   1:  PR[91,2] = PR[90,2] + 7.974;
   1:  PR[91,3] = PR[90,3] + 78.968;
   1:L PR[91] R[100]mm/sec CNT100;
   1:  PR[91,1] = PR[90,1] + 66.308;
   1:  PR[91,2] = PR[90,2] + 10.922;
   1:  PR[91,3] = PR[90,3] + 78.974;
   1:L PR[91] R[100]mm/sec CNT100;
   1:  PR[91,1] = PR[90,1] + 65.847;
   1:  PR[91,2] = PR[90,2] + 11.513;
   1:  PR[91,3] = PR[90,3] + 78.988;
   1:L PR[91] R[100]mm/sec CNT100;
   1:  PR[91,1] = PR[90,1] + 63.829;
   1:  PR[91,2] = PR[90,2] + 13.995;
   1:  PR[91,3] = PR[90,3] + 78.991;
   1:L PR[91] R[100]mm/sec CNT100;
   1:  PR[91,1] = PR[90,1] + 63.263;
   1:  PR[91,2] = PR[90,2] + 14.657;
   1:  PR[91,3] = PR[90,3] + 79.003;
   1:L PR[91] R[100]mm/sec CNT100;
   1:  PR[91,1] = PR[90,1] + 62.571;
   1:  PR[91,2] = PR[90,2] + 15.260;
   1:  PR[91,3] = PR[90,3] + 79.007;
   1:L PR[91] R[100]mm/sec CNT100;
   1:  PR[91,1] = PR[90,1] + 59.786;
   1:  PR[91,2] = PR[90,2] + 17.613;
   1:  PR[91,3] = PR[90,3] + 79.010;
   1:L PR[91] R[100]mm/sec CNT100;
   1:  PR[91,1] = PR[90,1] + 57.560;
   1:  PR[91,2] = PR[90,2] + 19.039;
   1:  PR[91,3] = PR[90,3] + 79.024;
   1:L PR[91] R[100]mm/sec CNT100;
   1:  PR[91,1] = PR[90,1] + 56.192;
   1:  PR[91,2] = PR[90,2] + 20.065;
   1:  PR[91,3] = PR[90,3] + 79.035;
   1:L PR[91] R[100]mm/sec CNT100;
   1:  PR[91,1] = PR[90,1] + 54.654;
   1:  PR[91,2] = PR[90,2] + 20.998;
   1:  PR[91,3] = PR[90,3] + 79.042;
   1:L PR[91] R[100]mm/sec CNT100;
   1:  PR[91,1] = PR[90,1] + 52.639;
   1:  PR[91,2] = PR[90,2] + 22.108;
   1:  PR[91,3] = PR[90,3] + 79.049;
   1:L PR[91] R[100]mm/sec CNT100;
   1:  PR[91,1] = PR[90,1] + 50.085;
   1:  PR[91,2] = PR[90,2] + 23.189;
   1:  PR[91,3] = PR[90,3] + 79.058;
   1:L PR[91] R[100]mm/sec CNT100;
   1:  PR[91,1] = PR[90,1] + 48.507;
   1:  PR[91,2] = PR[90,2] + 24.012;
   1:  PR[91,3] = PR[90,3] + 79.069;
   1:L PR[91] R[100]mm/sec CNT100;
   1:  PR[91,1] = PR[90,1] + 47.413;
   1:  PR[91,2] = PR[90,2] + 24.469;
   1:  PR[91,3] = PR[90,3] + 79.075;
   1:L PR[91] R[100]mm/sec CNT100;
   1:  PR[91,1] = PR[90,1] + 44.640;
   1:  PR[91,2] = PR[90,2] + 25.399;
   1:  PR[91,3] = PR[90,3] + 79.080;
   1:L PR[91] R[100]mm/sec CNT100;
   1:  PR[91,1] = PR[90,1] + 40.467;
   1:  PR[91,2] = PR[90,2] + 26.399;
   1:  PR[91,3] = PR[90,3] + 79.092;
   1:L PR[91] R[100]mm/sec CNT100;
   1:  PR[91,1] = PR[90,1] + 40.116;
   1:  PR[91,2] = PR[90,2] + 26.460;
   1:  PR[91,3] = PR[90,3] + 79.108;
   1:L PR[91] R[100]mm/sec CNT100;
   1:  PR[91,1] = PR[90,1] + 39.134;
   1:  PR[91,2] = PR[90,2] + 26.535;
   1:  PR[91,3] = PR[90,3] + 79.110;
   1:L PR[91] R[100]mm/sec CNT100;
   1:  PR[91,1] = PR[90,1] + 34.948;
   1:  PR[91,2] = PR[90,2] + 26.936;
   1:  PR[91,3] = PR[90,3] + 79.114;
   1:L PR[91] R[100]mm/sec CNT100;
   1:  PR[91,1] = PR[90,1] + 33.069;
   1:  PR[91,2] = PR[90,2] + 26.830;
   1:  PR[91,3] = PR[90,3] + 79.130;
   1:L PR[91] R[100]mm/sec CNT100;
   1:  PR[91,1] = PR[90,1] + 29.800;
   1:  PR[91,2] = PR[90,2] + 26.569;
   1:  PR[91,3] = PR[90,3] + 79.138;
   1:L PR[91] R[100]mm/sec CNT100;
   1:  PR[91,1] = PR[90,1] + 26.009;
   1:  PR[91,2] = PR[90,2] + 25.701;
   1:  PR[91,3] = PR[90,3] + 79.150;
   1:L PR[91] R[100]mm/sec CNT100;
   1:  PR[91,1] = PR[90,1] + 24.298;
   1:  PR[91,2] = PR[90,2] + 25.254;
   1:  PR[91,3] = PR[90,3] + 79.166;
   1:L PR[91] R[100]mm/sec CNT100;
   1:  PR[91,1] = PR[90,1] + 23.224;
   1:  PR[91,2] = PR[90,2] + 25.412;
   1:  PR[91,3] = PR[90,3] + 79.173;
   1:L PR[91] R[100]mm/sec CNT100;
   1:  PR[91,1] = PR[90,1] + 16.968;
   1:  PR[91,2] = PR[90,2] + 25.613;
   1:  PR[91,3] = PR[90,3] + 79.177;
   1:L PR[91] R[100]mm/sec CNT100;
   1:  PR[91,1] = PR[90,1] + 16.795;
   1:  PR[91,2] = PR[90,2] + 25.606;
   1:  PR[91,3] = PR[90,3] + 79.202;
   1:L PR[91] R[100]mm/sec CNT100;
   1:  PR[91,1] = PR[90,1] + 9.750;
   1:  PR[91,2] = PR[90,2] + 24.089;
   1:L PR[91] R[100]mm/sec CNT100;
   1:  PR[91,1] = PR[90,1] + 8.665;
   1:  PR[91,2] = PR[90,2] + 24.309;
   1:  PR[91,3] = PR[90,3] + 79.230;
   1:L PR[91] R[100]mm/sec CNT100;
   1:  PR[91,1] = PR[90,1] + 5.140;
   1:  PR[91,2] = PR[90,2] + 24.727;
   1:  PR[91,3] = PR[90,3] + 79.235;
   1:L PR[91] R[100]mm/sec CNT100;
   1:  PR[91,1] = PR[90,1] + 2.127;
   1:  PR[91,2] = PR[90,2] + 24.938;
   1:  PR[91,3] = PR[90,3] + 79.249;
   1:L PR[91] R[100]mm/sec CNT100;
   1:  PR[91,1] = PR[90,1] + -0.101;
   1:  PR[91,2] = PR[90,2] + 24.933;
   1:  PR[91,3] = PR[90,3] + 79.261;
   1:L PR[91] R[100]mm/sec CNT100;
   1:  PR[91,1] = PR[90,1] + -6.393;
   1:  PR[91,2] = PR[90,2] + 24.297;
   1:  PR[91,3] = PR[90,3] + 79.269;
   1:L PR[91] R[100]mm/sec CNT100;
   1:  PR[91,1] = PR[90,1] + -11.231;
   1:  PR[91,2] = PR[90,2] + 24.737;
   1:  PR[91,3] = PR[90,3] + 79.294;
   1:L PR[91] R[100]mm/sec CNT100;
   1:  PR[91,1] = PR[90,1] + -18.619;
   1:  PR[91,2] = PR[90,2] + 25.021;
   1:  PR[91,3] = PR[90,3] + 79.313;
   1:L PR[91] R[100]mm/sec CNT100;
   1:  PR[91,1] = PR[90,1] + -21.356;
   1:  PR[91,2] = PR[90,2] + 25.107;
   1:  PR[91,3] = PR[90,3] + 79.342;
   1:L PR[91] R[100]mm/sec CNT100;
   1:  PR[91,1] = PR[90,1] + -30.684;
   1:  PR[91,2] = PR[90,2] + 24.799;
   1:  PR[91,3] = PR[90,3] + 79.353;
   1:L PR[91] R[100]mm/sec CNT100;
   1:  PR[91,1] = PR[90,1] + -31.732;
   1:  PR[91,2] = PR[90,2] + 24.710;
   1:  PR[91,3] = PR[90,3] + 79.390;
   1:L PR[91] R[100]mm/sec CNT100;
   1:  PR[91,1] = PR[90,1] + -37.259;
   1:  PR[91,2] = PR[90,2] + 24.127;
   1:  PR[91,3] = PR[90,3] + 79.394;
   1:L PR[91] R[100]mm/sec CNT100;
   1:  PR[91,1] = PR[90,1] + -44.886;
   1:  PR[91,2] = PR[90,2] + 22.670;
   1:  PR[91,3] = PR[90,3] + 79.416;
   1:L PR[91] R[100]mm/sec CNT100;
   1:  PR[91,1] = PR[90,1] + -51.856;
   1:  PR[91,2] = PR[90,2] + 20.497;
   1:  PR[91,3] = PR[90,3] + 79.446;
   1:L PR[91] R[100]mm/sec CNT100;
   1:  PR[91,1] = PR[90,1] + -56.441;
   1:  PR[91,2] = PR[90,2] + 18.105;
   1:  PR[91,3] = PR[90,3] + 79.475;
   1:L PR[91] R[100]mm/sec CNT100;
   1:  PR[91] = PR[90];
   1:  PR[91,1] = PR[90,1] + -57.127;
   1:  PR[91,2] = PR[90,2] + 17.164;
   1:  PR[91,3] = PR[90,3] + 80.795;
   1:L PR[91] R[100]mm/sec CNT100;
   1:  PR[91,1] = PR[90,1] + -59.761;
   1:  PR[91,2] = PR[90,2] + 15.080;
   1:  PR[91,3] = PR[90,3] + 79.501;
   1:L PR[91] R[100]mm/sec CNT100;
   1:  PR[91,1] = PR[90,1] + -62.266;
   1:  PR[91,2] = PR[90,2] + 13.000;
   1:  PR[91,3] = PR[90,3] + 79.514;
   1:L PR[91] R[100]mm/sec CNT100;
   1:  PR[91,1] = PR[90,1] + -63.125;
   1:  PR[91,2] = PR[90,2] + 11.946;
   1:  PR[91,3] = PR[90,3] + 79.527;
   1:L PR[91] R[100]mm/sec CNT100;
   1:  PR[91,1] = PR[90,1] + -65.801;
   1:  PR[91,2] = PR[90,2] + 8.538;
   1:  PR[91,3] = PR[90,3] + 79.532;
   1:L PR[91] R[100]mm/sec CNT100;
   1:  PR[91,1] = PR[90,1] + -66.670;
   1:  PR[91,2] = PR[90,2] + 6.598;
   1:  PR[91,3] = PR[90,3] + 79.550;
   1:L PR[91] R[100]mm/sec CNT100;
   1:  PR[91,1] = PR[90,1] + -67.726;
   1:  PR[91,2] = PR[90,2] + 3.985;
   1:  PR[91,3] = PR[90,3] + 79.558;
   1:L PR[91] R[100]mm/sec CNT100;
   1:  PR[91,1] = PR[90,1] + -67.747;
   1:  PR[91,2] = PR[90,2] + 3.823;
   1:  PR[91,3] = PR[90,3] + 79.569;
   1:L PR[91] R[100]mm/sec CNT100;
   1:  PR[91,1] = PR[90,1] + -67.921;
   1:  PR[91,2] = PR[90,2] + 2.835;
   1:  PR[91,3] = PR[90,3] + 79.570;
   1:L PR[91] R[100]mm/sec CNT100;
   1:  PR[91,1] = PR[90,1] + -68.404;
   1:  PR[91,2] = PR[90,2] + -0.725;
   1:  PR[91,3] = PR[90,3] + 79.574;
   1:L PR[91] R[100]mm/sec CNT100;
   1:  PR[91,1] = PR[90,1] + -68.209;
   1:  PR[91,2] = PR[90,2] + -2.121;
   1:  PR[91,3] = PR[90,3] + 79.588;
   1:L PR[91] R[100]mm/sec CNT100;
   1:  PR[91,1] = PR[90,1] + -67.922;
   1:  PR[91,2] = PR[90,2] + -3.706;
   1:  PR[91,3] = PR[90,3] + 79.594;
   1:L PR[91] R[100]mm/sec CNT100;
   1:  PR[91,1] = PR[90,1] + -67.733;
   1:  PR[91,2] = PR[90,2] + -4.386;
   1:  PR[91,3] = PR[90,3] + 79.600;
   1:L PR[91] R[100]mm/sec CNT100;
   1:  PR[91,1] = PR[90,1] + -67.589;
   1:  PR[91,2] = PR[90,2] + -5.467;
   1:  PR[91,3] = PR[90,3] + 79.603;
   1:L PR[91] R[100]mm/sec CNT100;
   1:  PR[91,1] = PR[90,1] + -67.132;
   1:  PR[91,2] = PR[90,2] + -6.573;
   1:  PR[91,3] = PR[90,3] + 79.607;
   1:L PR[91] R[100]mm/sec CNT100;
   1:  PR[91,1] = PR[90,1] + -65.623;
   1:  PR[91,2] = PR[90,2] + -9.993;
   1:  PR[91,3] = PR[90,3] + 79.612;
   1:L PR[91] R[100]mm/sec CNT100;
   1:  PR[91,1] = PR[90,1] + -64.279;
   1:  PR[91,2] = PR[90,2] + -11.843;
   1:  PR[91,3] = PR[90,3] + 79.627;
   1:L PR[91] R[100]mm/sec CNT100;
   1:  PR[91,1] = PR[90,1] + -62.471;
   1:  PR[91,2] = PR[90,2] + -14.163;
   1:  PR[91,3] = PR[90,3] + 79.636;
   1:L PR[91] R[100]mm/sec CNT100;
   1:  PR[91,1] = PR[90,1] + -59.300;
   1:  PR[91,2] = PR[90,2] + -17.023;
   1:  PR[91,3] = PR[90,3] + 79.648;
   1:L PR[91] R[100]mm/sec CNT100;
   1:  PR[91,1] = PR[90,1] + -58.360;
   1:  PR[91,2] = PR[90,2] + -17.807;
   1:  PR[91,3] = PR[90,3] + 79.665;
   1:L PR[91] R[100]mm/sec CNT100;
   1:  PR[91,1] = PR[90,1] + -55.860;
   1:  PR[91,2] = PR[90,2] + -19.339;
   1:  PR[91,3] = PR[90,3] + 79.670;
   1:L PR[91] R[100]mm/sec CNT100;
   1:  PR[91,1] = PR[90,1] + -53.634;
   1:  PR[91,2] = PR[90,2] + -20.570;
   1:  PR[91,3] = PR[90,3] + 79.681;
   1:L PR[91] R[100]mm/sec CNT100;
   1:  PR[91,1] = PR[90,1] + -52.629;
   1:  PR[91,2] = PR[90,2] + -21.092;
   1:  PR[91,3] = PR[90,3] + 79.691;
   1:L PR[91] R[100]mm/sec CNT100;
   1:  PR[91,1] = PR[90,1] + -48.737;
   1:  PR[91,2] = PR[90,2] + -22.548;
   1:  PR[91,3] = PR[90,3] + 79.696;
   1:L PR[91] R[100]mm/sec CNT100;
   1:  PR[91,1] = PR[90,1] + -44.199;
   1:  PR[91,2] = PR[90,2] + -24.096;
   1:  PR[91,3] = PR[90,3] + 79.712;
   1:L PR[91] R[100]mm/sec CNT100;
   1:  PR[91,1] = PR[90,1] + -43.532;
   1:  PR[91,2] = PR[90,2] + -24.250;
   1:  PR[91,3] = PR[90,3] + 79.731;
   1:L PR[91] R[100]mm/sec CNT100;
   1:  PR[91,1] = PR[90,1] + -42.508;
   1:  PR[91,2] = PR[90,2] + -24.451;
   1:  PR[91,3] = PR[90,3] + 79.734;
   1:L PR[91] R[100]mm/sec CNT100;
   1:  PR[91,1] = PR[90,1] + -35.626;
   1:  PR[91,2] = PR[90,2] + -25.731;
   1:  PR[91,3] = PR[90,3] + 79.738;
   1:L PR[91] R[100]mm/sec CNT100;
   1:  PR[91,1] = PR[90,1] + -28.455;
   1:  PR[91,2] = PR[90,2] + -26.491;
   1:  PR[91,3] = PR[90,3] + 79.766;
   1:L PR[91] R[100]mm/sec CNT100;
   1:  PR[91,1] = PR[90,1] + -18.729;
   1:  PR[91,2] = PR[90,2] + -26.818;
   1:  PR[91,3] = PR[90,3] + 79.795;
   1:L PR[91] R[100]mm/sec CNT100;
   1:  PR[91,1] = PR[90,1] + -14.970;
   1:  PR[91,2] = PR[90,2] + -26.700;
   1:  PR[91,3] = PR[90,3] + 79.833;
   1:L PR[91] R[100]mm/sec CNT100;
   1:  PR[91,1] = PR[90,1] + -8.725;
   1:  PR[91,2] = PR[90,2] + -26.466;
   1:  PR[91,3] = PR[90,3] + 79.848;
   1:L PR[91] R[100]mm/sec CNT100;
   1:  PR[91,1] = PR[90,1] + -8.035;
   1:  PR[91,2] = PR[90,2] + -26.416;
   1:  PR[91,3] = PR[90,3] + 79.873;
   1:L PR[91] R[100]mm/sec CNT100;
   1:  PR[91,1] = PR[90,1] + -5.547;
   1:  PR[91,2] = PR[90,2] + -26.134;
   1:  PR[91,3] = PR[90,3] + 79.876;
   1:L PR[91] R[100]mm/sec CNT100;
   1:  PR[91,1] = PR[90,1] + -4.527;
   1:  PR[91,2] = PR[90,2] + -26.106;
   1:  PR[91,3] = PR[90,3] + 79.886;
   1:L PR[91] R[100]mm/sec CNT100;
   1:  PR[91,1] = PR[90,1] + -0.160;
   1:  PR[91,2] = PR[90,2] + -26.561;
   1:  PR[91,3] = PR[90,3] + 79.890;
   1:L PR[91] R[100]mm/sec CNT100;
   1:  PR[91,1] = PR[90,1] + 0.543;
   1:  PR[91,2] = PR[90,2] + -26.607;
   1:  PR[91,3] = PR[90,3] + 79.907;
   1:L PR[91] R[100]mm/sec CNT100;
   1:  PR[91,1] = PR[90,1] + 3.638;
   1:  PR[91,2] = PR[90,2] + -26.613;
   1:  PR[91,3] = PR[90,3] + 79.910;
   1:L PR[91] R[100]mm/sec CNT100;
   1:  PR[91,1] = PR[90,1] + 5.637;
   1:  PR[91,2] = PR[90,2] + -26.475;
   1:  PR[91,3] = PR[90,3] + 79.922;
   1:L PR[91] R[100]mm/sec CNT100;
   1:  PR[91,1] = PR[90,1] + 10.246;
   1:  PR[91,2] = PR[90,2] + -25.930;
   1:  PR[91,3] = PR[90,3] + 79.930;
   1:L PR[91] R[100]mm/sec CNT100;
   1:  PR[91,1] = PR[90,1] + 16.533;
   1:  PR[91,2] = PR[90,2] + -27.222;
   1:  PR[91,3] = PR[90,3] + 79.949;
   1:L PR[91] R[100]mm/sec CNT100;
   1:  PR[91,1] = PR[90,1] + 16.683;
   1:  PR[91,2] = PR[90,2] + -27.244;
   1:  PR[91,3] = PR[90,3] + 79.974;
   1:L PR[91] R[100]mm/sec CNT100;
   1:  PR[91,1] = PR[90,1] + 23.285;
   1:  PR[91,2] = PR[90,2] + -27.027;
   1:  PR[91,3] = PR[90,3] + 79.975;
   1:L PR[91] R[100]mm/sec CNT100;
   1:  PR[91,1] = PR[90,1] + 23.841;
   1:  PR[91,2] = PR[90,2] + -26.952;
   1:  PR[91,3] = PR[90,3] + 80.001;
   1:L PR[91] R[100]mm/sec CNT100;
   1:  PR[91,1] = PR[90,1] + 24.558;
   1:  PR[91,2] = PR[90,2] + -27.139;
   1:  PR[91,3] = PR[90,3] + 80.003;
   1:L PR[91] R[100]mm/sec CNT100;
   1:  PR[91,1] = PR[90,1] + 29.428;
   1:  PR[91,2] = PR[90,2] + -28.254;
   1:  PR[91,3] = PR[90,3] + 80.006;
   1:L PR[91] R[100]mm/sec CNT100;
   1:  PR[91,1] = PR[90,1] + 31.477;
   1:  PR[91,2] = PR[90,2] + -28.418;
   1:  PR[91,3] = PR[90,3] + 80.026;
   1:L PR[91] R[100]mm/sec CNT100;
   1:  PR[91,1] = PR[90,1] + 34.612;
   1:  PR[91,2] = PR[90,2] + -28.595;
   1:  PR[91,3] = PR[90,3] + 80.034;
   1:L PR[91] R[100]mm/sec CNT100;
   1:  PR[91,1] = PR[90,1] + 39.040;
   1:  PR[91,2] = PR[90,2] + -28.171;
   1:  PR[91,3] = PR[90,3] + 80.047;
   1:L PR[91] R[100]mm/sec CNT100;
   1:  PR[91,1] = PR[90,1] + 39.704;
   1:  PR[91,2] = PR[90,2] + -28.096;
   1:  PR[91,3] = PR[90,3] + 80.064;
   1:L PR[91] R[100]mm/sec CNT100;
   1:  PR[91,1] = PR[90,1] + 41.112;
   1:  PR[91,2] = PR[90,2] + -27.706;
   1:  PR[91,3] = PR[90,3] + 80.067;
   1:L PR[91] R[100]mm/sec CNT100;
   1:  PR[91,1] = PR[90,1] + 44.509;
   1:  PR[91,2] = PR[90,2] + -26.892;
   1:  PR[91,3] = PR[90,3] + 80.073;
   1:L PR[91] R[100]mm/sec CNT100;
   1:  PR[91,1] = PR[90,1] + 46.070;
   1:  PR[91,2] = PR[90,2] + -26.368;
   1:  PR[91,3] = PR[90,3] + 80.087;
   1:L PR[91] R[100]mm/sec CNT100;
   1:  PR[91,1] = PR[90,1] + 48.476;
   1:  PR[91,2] = PR[90,2] + -25.364;
   1:  PR[91,3] = PR[90,3] + 80.093;
   1:L PR[91] R[100]mm/sec CNT100;
   1:  PR[91,1] = PR[90,1] + 51.725;
   1:  PR[91,2] = PR[90,2] + -23.668;
   1:  PR[91,3] = PR[90,3] + 80.104;
   1:L PR[91] R[100]mm/sec CNT100;
   1:  PR[91,1] = PR[90,1] + 52.139;
   1:  PR[91,2] = PR[90,2] + -23.493;
   1:  PR[91,3] = PR[90,3] + 80.118;
   1:L PR[91] R[100]mm/sec CNT100;
   1:  PR[91,1] = PR[90,1] + 52.374;
   1:  PR[91,2] = PR[90,2] + -23.364;
   1:  PR[91,3] = PR[90,3] + 80.120;
   1:L PR[91] R[100]mm/sec CNT100;
   1:  PR[91,1] = PR[90,1] + 55.803;
   1:  PR[91,2] = PR[90,2] + -21.284;
   1:  PR[91,3] = PR[90,3] + 80.121;
   1:L PR[91] R[100]mm/sec CNT100;
   1:  PR[91,1] = PR[90,1] + 58.756;
   1:  PR[91,2] = PR[90,2] + -19.070;
   1:  PR[91,3] = PR[90,3] + 80.137;
   1:L PR[91] R[100]mm/sec CNT100;
   1:  PR[91,1] = PR[90,1] + 58.864;
   1:  PR[91,2] = PR[90,2] + -19.001;
   1:  PR[91,3] = PR[90,3] + 80.152;
   1:L PR[91] R[100]mm/sec CNT100;
   1:  PR[91,1] = PR[90,1] + 62.286;
   1:  PR[91,2] = PR[90,2] + -16.027;
   1:L PR[91] R[100]mm/sec CNT100;
   1:  PR[91,1] = PR[90,1] + 65.022;
   1:  PR[91,2] = PR[90,2] + -12.827;
   1:  PR[91,3] = PR[90,3] + 80.170;
   1:L PR[91] R[100]mm/sec CNT100;
   1:  PR[91,1] = PR[90,1] + 65.182;
   1:  PR[91,2] = PR[90,2] + -12.628;
   1:  PR[91,3] = PR[90,3] + 80.187;
   1:L PR[91] R[100]mm/sec CNT100;
   1:  PR[91,1] = PR[90,1] + 67.131;
   1:  PR[91,2] = PR[90,2] + -9.121;
   1:  PR[91,3] = PR[90,3] + 80.188;
   1:L PR[91] R[100]mm/sec CNT100;
   1:  PR[91,1] = PR[90,1] + 67.452;
   1:  PR[91,2] = PR[90,2] + -8.389;
   1:  PR[91,3] = PR[90,3] + 80.204;
   1:L PR[91] R[100]mm/sec CNT100;
   1:  PR[91,1] = PR[90,1] + 68.507;
   1:  PR[91,2] = PR[90,2] + -5.114;
   1:  PR[91,3] = PR[90,3] + 80.207;
   1:L PR[91] R[100]mm/sec CNT100;
   1:  PR[91,1] = PR[90,1] + 68.691;
   1:  PR[91,2] = PR[90,2] + -3.827;
   1:  PR[91,3] = PR[90,3] + 80.221;
   1:L PR[91] R[100]mm/sec CNT100;
   1:  PR[91,1] = PR[90,1] + 69.013;
   1:  PR[91,2] = PR[90,2] + -0.768;
   1:  PR[91,3] = PR[90,3] + 80.226;
   1:L PR[91] R[100]mm/sec CNT100;
   1:  PR[91,1] = PR[90,1] + 68.818;
   1:  PR[91,2] = PR[90,2] + 0.583;
   1:  PR[91,3] = PR[90,3] + 80.238;
   1:L PR[91] R[100]mm/sec CNT100;
   1:  PR[91,1] = PR[90,1] + 68.495;
   1:  PR[91,2] = PR[90,2] + 3.691;
   1:  PR[91,3] = PR[90,3] + 80.243;
   1:L PR[91] R[100]mm/sec CNT100;
   1:  PR[91,1] = PR[90,1] + 67.452;
   1:  PR[91,2] = PR[90,2] + 6.930;
   1:  PR[91,3] = PR[90,3] + 80.256;
   1:L PR[91] R[100]mm/sec CNT100;
   1:  PR[91,1] = PR[90,1] + 67.132;
   1:  PR[91,2] = PR[90,2] + 7.661;
   1:  PR[91,3] = PR[90,3] + 80.269;
   1:L PR[91] R[100]mm/sec CNT100;
   1:  PR[91,1] = PR[90,1] + 65.182;
   1:  PR[91,2] = PR[90,2] + 11.169;
   1:  PR[91,3] = PR[90,3] + 80.272;
   1:L PR[91] R[100]mm/sec CNT100;
   1:  PR[91,1] = PR[90,1] + 65.022;
   1:  PR[91,2] = PR[90,2] + 11.368;
   1:  PR[91,3] = PR[90,3] + 80.288;
   1:L PR[91] R[100]mm/sec CNT100;
   1:  PR[91,1] = PR[90,1] + 62.286;
   1:  PR[91,2] = PR[90,2] + 14.568;
   1:  PR[91,3] = PR[90,3] + 80.289;
   1:L PR[91] R[100]mm/sec CNT100;
   1:  PR[91,1] = PR[90,1] + 58.864;
   1:  PR[91,2] = PR[90,2] + 17.542;
   1:  PR[91,3] = PR[90,3] + 80.306;
   1:L PR[91] R[100]mm/sec CNT100;
   1:  PR[91,1] = PR[90,1] + 58.756;
   1:  PR[91,2] = PR[90,2] + 17.612;
   1:  PR[91,3] = PR[90,3] + 80.324;
   1:L PR[91] R[100]mm/sec CNT100;
   1:  PR[91,1] = PR[90,1] + 55.803;
   1:  PR[91,2] = PR[90,2] + 19.826;
   1:  PR[91,3] = PR[90,3] + 80.325;
   1:L PR[91] R[100]mm/sec CNT100;
   1:  PR[91,1] = PR[90,1] + 52.374;
   1:  PR[91,2] = PR[90,2] + 21.905;
   1:  PR[91,3] = PR[90,3] + 80.339;
   1:L PR[91] R[100]mm/sec CNT100;
   1:  PR[91,1] = PR[90,1] + 52.139;
   1:  PR[91,2] = PR[90,2] + 22.034;
   1:  PR[91,3] = PR[90,3] + 80.355;
   1:L PR[91] R[100]mm/sec CNT100;
   1:  PR[91,1] = PR[90,1] + 51.725;
   1:  PR[91,2] = PR[90,2] + 22.209;
   1:  PR[91,3] = PR[90,3] + 80.356;
   1:L PR[91] R[100]mm/sec CNT100;
   1:  PR[91,1] = PR[90,1] + 48.476;
   1:  PR[91,2] = PR[90,2] + 23.905;
   1:  PR[91,3] = PR[90,3] + 80.358;
   1:L PR[91] R[100]mm/sec CNT100;
   1:  PR[91,1] = PR[90,1] + 46.070;
   1:  PR[91,2] = PR[90,2] + 24.909;
   1:  PR[91,3] = PR[90,3] + 80.373;
   1:L PR[91] R[100]mm/sec CNT100;
   1:  PR[91,1] = PR[90,1] + 44.509;
   1:  PR[91,2] = PR[90,2] + 25.434;
   1:  PR[91,3] = PR[90,3] + 80.383;
   1:L PR[91] R[100]mm/sec CNT100;
   1:  PR[91,1] = PR[90,1] + 41.112;
   1:  PR[91,2] = PR[90,2] + 26.248;
   1:  PR[91,3] = PR[90,3] + 80.390;
   1:L PR[91] R[100]mm/sec CNT100;
   1:  PR[91,1] = PR[90,1] + 39.704;
   1:  PR[91,2] = PR[90,2] + 26.637;
   1:  PR[91,3] = PR[90,3] + 80.403;
   1:L PR[91] R[100]mm/sec CNT100;
   1:  PR[91,1] = PR[90,1] + 39.040;
   1:  PR[91,2] = PR[90,2] + 26.712;
   1:  PR[91,3] = PR[90,3] + 80.409;
   1:L PR[91] R[100]mm/sec CNT100;
   1:  PR[91,1] = PR[90,1] + 34.612;
   1:  PR[91,2] = PR[90,2] + 27.136;
   1:  PR[91,3] = PR[90,3] + 80.412;
   1:L PR[91] R[100]mm/sec CNT100;
   1:  PR[91,1] = PR[90,1] + 31.477;
   1:  PR[91,2] = PR[90,2] + 26.959;
   1:  PR[91,3] = PR[90,3] + 80.430;
   1:L PR[91] R[100]mm/sec CNT100;
   1:  PR[91,1] = PR[90,1] + 29.428;
   1:  PR[91,2] = PR[90,2] + 26.796;
   1:  PR[91,3] = PR[90,3] + 80.442;
   1:L PR[91] R[100]mm/sec CNT100;
   1:  PR[91,1] = PR[90,1] + 24.558;
   1:  PR[91,2] = PR[90,2] + 25.680;
   1:  PR[91,3] = PR[90,3] + 80.450;
   1:L PR[91] R[100]mm/sec CNT100;
   1:  PR[91,1] = PR[90,1] + 23.841;
   1:  PR[91,2] = PR[90,2] + 25.493;
   1:  PR[91,3] = PR[90,3] + 80.470;
   1:L PR[91] R[100]mm/sec CNT100;
   1:  PR[91,1] = PR[90,1] + 23.285;
   1:  PR[91,2] = PR[90,2] + 25.568;
   1:  PR[91,3] = PR[90,3] + 80.473;
   1:L PR[91] R[100]mm/sec CNT100;
   1:  PR[91,1] = PR[90,1] + 16.683;
   1:  PR[91,2] = PR[90,2] + 25.785;
   1:  PR[91,3] = PR[90,3] + 80.475;
   1:L PR[91] R[100]mm/sec CNT100;
   1:  PR[91,1] = PR[90,1] + 16.533;
   1:  PR[91,2] = PR[90,2] + 25.763;
   1:  PR[91,3] = PR[90,3] + 80.501;
   1:L PR[91] R[100]mm/sec CNT100;
   1:  PR[91,1] = PR[90,1] + 10.246;
   1:  PR[91,2] = PR[90,2] + 24.471;
   1:  PR[91,3] = PR[90,3] + 80.502;
   1:L PR[91] R[100]mm/sec CNT100;
   1:  PR[91,1] = PR[90,1] + 5.647;
   1:  PR[91,2] = PR[90,2] + 25.015;
   1:  PR[91,3] = PR[90,3] + 80.528;
   1:L PR[91] R[100]mm/sec CNT100;
   1:  PR[91,1] = PR[90,1] + 3.650;
   1:  PR[91,2] = PR[90,2] + 25.155;
   1:  PR[91,3] = PR[90,3] + 80.546;
   1:L PR[91] R[100]mm/sec CNT100;
   1:  PR[91,1] = PR[90,1] + 0.598;
   1:  PR[91,2] = PR[90,2] + 25.148;
   1:  PR[91,3] = PR[90,3] + 80.554;
   1:L PR[91] R[100]mm/sec CNT100;
   1:  PR[91,1] = PR[90,1] + -4.527;
   1:  PR[91,2] = PR[90,2] + 24.630;
   1:  PR[91,3] = PR[90,3] + 80.566;
   1:L PR[91] R[100]mm/sec CNT100;
   1:  PR[91,1] = PR[90,1] + -8.480;
   1:  PR[91,2] = PR[90,2] + 24.990;
   1:  PR[91,3] = PR[90,3] + 80.586;
   1:L PR[91] R[100]mm/sec CNT100;
   1:  PR[91,1] = PR[90,1] + -14.972;
   1:  PR[91,2] = PR[90,2] + 25.241;
   1:  PR[91,3] = PR[90,3] + 80.602;
   1:L PR[91] R[100]mm/sec CNT100;
   1:  PR[91,1] = PR[90,1] + -18.729;
   1:  PR[91,2] = PR[90,2] + 25.359;
   1:  PR[91,3] = PR[90,3] + 80.628;
   1:L PR[91] R[100]mm/sec CNT100;
   1:  PR[91,1] = PR[90,1] + -28.456;
   1:  PR[91,2] = PR[90,2] + 25.032;
   1:  PR[91,3] = PR[90,3] + 80.643;
   1:L PR[91] R[100]mm/sec CNT100;
   1:  PR[91,1] = PR[90,1] + -35.694;
   1:  PR[91,2] = PR[90,2] + 24.272;
   1:  PR[91,3] = PR[90,3] + 80.682;
   1:L PR[91] R[100]mm/sec CNT100;
   1:  PR[91,1] = PR[90,1] + -43.684;
   1:  PR[91,2] = PR[90,2] + 22.754;
   1:  PR[91,3] = PR[90,3] + 80.710;
   1:L PR[91] R[100]mm/sec CNT100;
   1:  PR[91,1] = PR[90,1] + -47.455;
   1:  PR[91,2] = PR[90,2] + 21.581;
   1:  PR[91,3] = PR[90,3] + 80.743;
   1:L PR[91] R[100]mm/sec CNT100;
   1:  PR[91,1] = PR[90,1] + -50.593;
   1:  PR[91,2] = PR[90,2] + 20.532;
   1:  PR[91,3] = PR[90,3] + 80.758;
   1:L PR[91] R[100]mm/sec CNT100;
   1:  PR[91,1] = PR[90,1] + -52.958;
   1:  PR[91,2] = PR[90,2] + 19.392;
   1:  PR[91,3] = PR[90,3] + 80.772;
   1:L PR[91] R[100]mm/sec CNT100;
   1:  PR[91,1] = PR[90,1] + -55.848;
   1:  PR[91,2] = PR[90,2] + 17.879;
   1:  PR[91,3] = PR[90,3] + 80.782;
   1:L PR[91] R[100]mm/sec CNT100;
   1:  PR[91] = PR[90];
   1:  PR[91,1] = PR[90,1] + -59.097;
   1:  PR[91,2] = PR[90,2] + 14.724;
   1:  PR[91,3] = PR[90,3] + 82.095;
   1:L PR[91] R[100]mm/sec CNT100;
   1:  PR[91,1] = PR[90,1] + -60.961;
   1:  PR[91,2] = PR[90,2] + 13.177;
   1:  PR[91,3] = PR[90,3] + 80.812;
   1:L PR[91] R[100]mm/sec CNT100;
   1:  PR[91,1] = PR[90,1] + -62.361;
   1:  PR[91,2] = PR[90,2] + 11.459;
   1:  PR[91,3] = PR[90,3] + 80.822;
   1:L PR[91] R[100]mm/sec CNT100;
   1:  PR[91,1] = PR[90,1] + -64.566;
   1:  PR[91,2] = PR[90,2] + 8.651;
   1:  PR[91,3] = PR[90,3] + 80.831;
   1:L PR[91] R[100]mm/sec CNT100;
   1:  PR[91,1] = PR[90,1] + -64.934;
   1:  PR[91,2] = PR[90,2] + 7.850;
   1:  PR[91,3] = PR[90,3] + 80.845;
   1:L PR[91] R[100]mm/sec CNT100;
   1:  PR[91,1] = PR[90,1] + -66.656;
   1:  PR[91,2] = PR[90,2] + 3.986;
   1:  PR[91,3] = PR[90,3] + 80.849;
   1:L PR[91] R[100]mm/sec CNT100;
   1:  PR[91,1] = PR[90,1] + -67.348;
   1:  PR[91,2] = PR[90,2] + -0.728;
   1:  PR[91,3] = PR[90,3] + 80.866;
   1:L PR[91] R[100]mm/sec CNT100;
   1:  PR[91,1] = PR[90,1] + -66.993;
   1:  PR[91,2] = PR[90,2] + -2.684;
   1:  PR[91,3] = PR[90,3] + 80.885;
   1:L PR[91] R[100]mm/sec CNT100;
   1:  PR[91,1] = PR[90,1] + -66.707;
   1:  PR[91,2] = PR[90,2] + -3.713;
   1:  PR[91,3] = PR[90,3] + 80.893;
   1:L PR[91] R[100]mm/sec CNT100;
   1:  PR[91,1] = PR[90,1] + -66.475;
   1:  PR[91,2] = PR[90,2] + -5.456;
   1:  PR[91,3] = PR[90,3] + 80.897;
   1:L PR[91] R[100]mm/sec CNT100;
   1:  PR[91,1] = PR[90,1] + -65.707;
   1:  PR[91,2] = PR[90,2] + -7.317;
   1:  PR[91,3] = PR[90,3] + 80.904;
   1:L PR[91] R[100]mm/sec CNT100;
   1:  PR[91,1] = PR[90,1] + -64.534;
   1:  PR[91,2] = PR[90,2] + -9.975;
   1:  PR[91,3] = PR[90,3] + 80.912;
   1:L PR[91] R[100]mm/sec CNT100;
   1:  PR[91,1] = PR[90,1] + -62.639;
   1:  PR[91,2] = PR[90,2] + -12.585;
   1:  PR[91,3] = PR[90,3] + 80.924;
   1:L PR[91] R[100]mm/sec CNT100;
   1:  PR[91,1] = PR[90,1] + -61.422;
   1:  PR[91,2] = PR[90,2] + -14.146;
   1:  PR[91,3] = PR[90,3] + 80.937;
   1:L PR[91] R[100]mm/sec CNT100;
   1:  PR[91,1] = PR[90,1] + -57.445;
   1:  PR[91,2] = PR[90,2] + -17.734;
   1:  PR[91,3] = PR[90,3] + 80.945;
   1:L PR[91] R[100]mm/sec CNT100;
   1:  PR[91,1] = PR[90,1] + -57.362;
   1:  PR[91,2] = PR[90,2] + -17.803;
   1:  PR[91,3] = PR[90,3] + 80.967;
   1:L PR[91] R[100]mm/sec CNT100;
   1:  PR[91,1] = PR[90,1] + -56.971;
   1:  PR[91,2] = PR[90,2] + -18.043;
   1:L PR[91] R[100]mm/sec CNT100;
   1:  PR[91,1] = PR[90,1] + -52.816;
   1:  PR[91,2] = PR[90,2] + -20.339;
   1:  PR[91,3] = PR[90,3] + 80.969;
   1:L PR[91] R[100]mm/sec CNT100;
   1:  PR[91,1] = PR[90,1] + -50.855;
   1:  PR[91,2] = PR[90,2] + -21.359;
   1:  PR[91,3] = PR[90,3] + 80.988;
   1:L PR[91] R[100]mm/sec CNT100;
   1:  PR[91,1] = PR[90,1] + -47.969;
   1:  PR[91,2] = PR[90,2] + -22.438;
   1:  PR[91,3] = PR[90,3] + 80.997;
   1:L PR[91] R[100]mm/sec CNT100;
   1:  PR[91,1] = PR[90,1] + -43.135;
   1:  PR[91,2] = PR[90,2] + -24.088;
   1:  PR[91,3] = PR[90,3] + 81.009;
   1:L PR[91] R[100]mm/sec CNT100;
   1:  PR[91,1] = PR[90,1] + -42.305;
   1:  PR[91,2] = PR[90,2] + -24.336;
   1:  PR[91,3] = PR[90,3] + 81.030;
   1:L PR[91] R[100]mm/sec CNT100;
   1:  PR[91,1] = PR[90,1] + -40.753;
   1:  PR[91,2] = PR[90,2] + -24.637;
   1:  PR[91,3] = PR[90,3] + 81.033;
   1:L PR[91] R[100]mm/sec CNT100;
   1:  PR[91,1] = PR[90,1] + -34.092;
   1:  PR[91,2] = PR[90,2] + -25.875;
   1:  PR[91,3] = PR[90,3] + 81.039;
   1:L PR[91] R[100]mm/sec CNT100;
   1:  PR[91,1] = PR[90,1] + -25.910;
   1:  PR[91,2] = PR[90,2] + -26.735;
   1:  PR[91,3] = PR[90,3] + 81.067;
   1:L PR[91] R[100]mm/sec CNT100;
   1:  PR[91,1] = PR[90,1] + -16.101;
   1:  PR[91,2] = PR[90,2] + -27.071;
   1:  PR[91,3] = PR[90,3] + 81.100;
   1:L PR[91] R[100]mm/sec CNT100;
   1:  PR[91,1] = PR[90,1] + -11.322;
   1:  PR[91,2] = PR[90,2] + -26.920;
   1:  PR[91,3] = PR[90,3] + 81.139;
   1:L PR[91] R[100]mm/sec CNT100;
   1:  PR[91,1] = PR[90,1] + -6.014;
   1:  PR[91,2] = PR[90,2] + -26.721;
   1:  PR[91,3] = PR[90,3] + 81.158;
   1:L PR[91] R[100]mm/sec CNT100;
   1:  PR[91,1] = PR[90,1] + -5.208;
   1:  PR[91,2] = PR[90,2] + -26.663;
   1:  PR[91,3] = PR[90,3] + 81.180;
   1:L PR[91] R[100]mm/sec CNT100;
   1:  PR[91,1] = PR[90,1] + -3.478;
   1:  PR[91,2] = PR[90,2] + -26.467;
   1:  PR[91,3] = PR[90,3] + 81.183;
   1:L PR[91] R[100]mm/sec CNT100;
   1:  PR[91,1] = PR[90,1] + -2.707;
   1:  PR[91,2] = PR[90,2] + -26.446;
   1:  PR[91,3] = PR[90,3] + 81.190;
   1:L PR[91] R[100]mm/sec CNT100;
   1:  PR[91,1] = PR[90,1] + 0.335;
   1:  PR[91,2] = PR[90,2] + -26.763;
   1:  PR[91,3] = PR[90,3] + 81.193;
   1:L PR[91] R[100]mm/sec CNT100;
   1:  PR[91,1] = PR[90,1] + 1.244;
   1:  PR[91,2] = PR[90,2] + -26.822;
   1:  PR[91,3] = PR[90,3] + 81.205;
   1:L PR[91] R[100]mm/sec CNT100;
   1:  PR[91,1] = PR[90,1] + 5.167;
   1:  PR[91,2] = PR[90,2] + -26.830;
   1:  PR[91,3] = PR[90,3] + 81.209;
   1:L PR[91] R[100]mm/sec CNT100;
   1:  PR[91,1] = PR[90,1] + 6.150;
   1:  PR[91,2] = PR[90,2] + -26.762;
   1:  PR[91,3] = PR[90,3] + 81.225;
   1:L PR[91] R[100]mm/sec CNT100;
   1:  PR[91,1] = PR[90,1] + 8.363;
   1:  PR[91,2] = PR[90,2] + -26.500;
   1:  PR[91,3] = PR[90,3] + 81.229;
   1:L PR[91] R[100]mm/sec CNT100;
   1:  PR[91,1] = PR[90,1] + 10.803;
   1:  PR[91,2] = PR[90,2] + -26.256;
   1:  PR[91,3] = PR[90,3] + 81.238;
   1:L PR[91] R[100]mm/sec CNT100;
   1:  PR[91,1] = PR[90,1] + 15.320;
   1:  PR[91,2] = PR[90,2] + -27.185;
   1:  PR[91,3] = PR[90,3] + 81.248;
   1:L PR[91] R[100]mm/sec CNT100;
   1:  PR[91,1] = PR[90,1] + 16.175;
   1:  PR[91,2] = PR[90,2] + -27.328;
   1:  PR[91,3] = PR[90,3] + 81.266;
   1:L PR[91] R[100]mm/sec CNT100;
   1:  PR[91,1] = PR[90,1] + 16.871;
   1:  PR[91,2] = PR[90,2] + -27.413;
   1:  PR[91,3] = PR[90,3] + 81.270;
   1:L PR[91] R[100]mm/sec CNT100;
   1:  PR[91,1] = PR[90,1] + 23.534;
   1:  PR[91,2] = PR[90,2] + -27.191;
   1:  PR[91,3] = PR[90,3] + 81.272;
   1:L PR[91] R[100]mm/sec CNT100;
   1:  PR[91,1] = PR[90,1] + 26.132;
   1:  PR[91,2] = PR[90,2] + -27.811;
   1:  PR[91,3] = PR[90,3] + 81.299;
   1:L PR[91] R[100]mm/sec CNT100;
   1:  PR[91,1] = PR[90,1] + 29.056;
   1:  PR[91,2] = PR[90,2] + -28.481;
   1:  PR[91,3] = PR[90,3] + 81.310;
   1:L PR[91] R[100]mm/sec CNT100;
   1:  PR[91,1] = PR[90,1] + 29.886;
   1:  PR[91,2] = PR[90,2] + -28.547;
   1:  PR[91,3] = PR[90,3] + 81.322;
   1:L PR[91] R[100]mm/sec CNT100;
   1:  PR[91,1] = PR[90,1] + 34.276;
   1:  PR[91,2] = PR[90,2] + -28.794;
   1:  PR[91,3] = PR[90,3] + 81.325;
   1:L PR[91] R[100]mm/sec CNT100;
   1:  PR[91,1] = PR[90,1] + 37.303;
   1:  PR[91,2] = PR[90,2] + -28.504;
   1:  PR[91,3] = PR[90,3] + 81.343;
   1:L PR[91] R[100]mm/sec CNT100;
   1:  PR[91,1] = PR[90,1] + 39.402;
   1:  PR[91,2] = PR[90,2] + -28.267;
   1:  PR[91,3] = PR[90,3] + 81.355;
   1:L PR[91] R[100]mm/sec CNT100;
   1:  PR[91,1] = PR[90,1] + 43.418;
   1:  PR[91,2] = PR[90,2] + -27.157;
   1:  PR[91,3] = PR[90,3] + 81.364;
   1:L PR[91] R[100]mm/sec CNT100;
   1:  PR[91,1] = PR[90,1] + 44.378;
   1:  PR[91,2] = PR[90,2] + -26.927;
   1:  PR[91,3] = PR[90,3] + 81.381;
   1:L PR[91] R[100]mm/sec CNT100;
   1:  PR[91,1] = PR[90,1] + 44.728;
   1:  PR[91,2] = PR[90,2] + -26.809;
   1:  PR[91,3] = PR[90,3] + 81.385;
   1:L PR[91] R[100]mm/sec CNT100;
   1:  PR[91,1] = PR[90,1] + 48.444;
   1:  PR[91,2] = PR[90,2] + -25.257;
   1:  PR[91,3] = PR[90,3] + 81.386;
   1:L PR[91] R[100]mm/sec CNT100;
   1:  PR[91,1] = PR[90,1] + 50.965;
   1:  PR[91,2] = PR[90,2] + -23.942;
   1:  PR[91,3] = PR[90,3] + 81.402;
   1:L PR[91] R[100]mm/sec CNT100;
   1:  PR[91,1] = PR[90,1] + 51.821;
   1:  PR[91,2] = PR[90,2] + -23.403;
   1:  PR[91,3] = PR[90,3] + 81.414;
   1:L PR[91] R[100]mm/sec CNT100;
   1:  PR[91,1] = PR[90,1] + 53.101;
   1:  PR[91,2] = PR[90,2] + -22.447;
   1:  PR[91,3] = PR[90,3] + 81.418;
   1:L PR[91] R[100]mm/sec CNT100;
   1:  PR[91,1] = PR[90,1] + 55.414;
   1:  PR[91,2] = PR[90,2] + -21.045;
   1:  PR[91,3] = PR[90,3] + 81.424;
   1:L PR[91] R[100]mm/sec CNT100;
   1:  PR[91,1] = PR[90,1] + 57.005;
   1:  PR[91,2] = PR[90,2] + -19.852;
   1:  PR[91,3] = PR[90,3] + 81.435;
   1:L PR[91] R[100]mm/sec CNT100;
   1:  PR[91,1] = PR[90,1] + 58.345;
   1:  PR[91,2] = PR[90,2] + -18.719;
   1:  PR[91,3] = PR[90,3] + 81.443;
   1:L PR[91] R[100]mm/sec CNT100;
   1:  PR[91,1] = PR[90,1] + 59.721;
   1:  PR[91,2] = PR[90,2] + -17.321;
   1:  PR[91,3] = PR[90,3] + 81.450;
   1:L PR[91] R[100]mm/sec CNT100;
   1:  PR[91,1] = PR[90,1] + 61.308;
   1:  PR[91,2] = PR[90,2] + -15.938;
   1:  PR[91,3] = PR[90,3] + 81.458;
   1:L PR[91] R[100]mm/sec CNT100;
   1:  PR[91,1] = PR[90,1] + 62.644;
   1:  PR[91,2] = PR[90,2] + -14.376;
   1:  PR[91,3] = PR[90,3] + 81.466;
   1:L PR[91] R[100]mm/sec CNT100;
   1:  PR[91,1] = PR[90,1] + 64.150;
   1:  PR[91,2] = PR[90,2] + -12.560;
   1:  PR[91,3] = PR[90,3] + 81.475;
   1:L PR[91] R[100]mm/sec CNT100;
   1:  PR[91,1] = PR[90,1] + 66.017;
   1:  PR[91,2] = PR[90,2] + -9.345;
   1:  PR[91,3] = PR[90,3] + 81.484;
   1:L PR[91] R[100]mm/sec CNT100;
   1:  PR[91,1] = PR[90,1] + 66.304;
   1:  PR[91,2] = PR[90,2] + -8.829;
   1:  PR[91,3] = PR[90,3] + 81.499;
   1:L PR[91] R[100]mm/sec CNT100;
   1:  PR[91,1] = PR[90,1] + 67.558;
   1:  PR[91,2] = PR[90,2] + -4.939;
   1:  PR[91,3] = PR[90,3] + 81.501;
   1:L PR[91] R[100]mm/sec CNT100;
   1:  PR[91,1] = PR[90,1] + 67.624;
   1:  PR[91,2] = PR[90,2] + -4.472;
   1:  PR[91,3] = PR[90,3] + 81.518;
   1:L PR[91] R[100]mm/sec CNT100;
   1:  PR[91,1] = PR[90,1] + 68.015;
   1:  PR[91,2] = PR[90,2] + -0.768;
   1:  PR[91,3] = PR[90,3] + 81.520;
   1:L PR[91] R[100]mm/sec CNT100;
   1:  PR[91,1] = PR[90,1] + 67.931;
   1:  PR[91,2] = PR[90,2] + -0.182;
   1:  PR[91,3] = PR[90,3] + 81.535;
   1:L PR[91] R[100]mm/sec CNT100;
   1:  PR[91,1] = PR[90,1] + 67.546;
   1:  PR[91,2] = PR[90,2] + 3.516;
   1:  PR[91,3] = PR[90,3] + 81.537;
   1:L PR[91] R[100]mm/sec CNT100;
   1:  PR[91,1] = PR[90,1] + 66.304;
   1:  PR[91,2] = PR[90,2] + 7.370;
   1:  PR[91,3] = PR[90,3] + 81.552;
   1:L PR[91] R[100]mm/sec CNT100;
   1:  PR[91,1] = PR[90,1] + 66.017;
   1:  PR[91,2] = PR[90,2] + 7.887;
   1:  PR[91,3] = PR[90,3] + 81.568;
   1:L PR[91] R[100]mm/sec CNT100;
   1:  PR[91,1] = PR[90,1] + 64.150;
   1:  PR[91,2] = PR[90,2] + 11.101;
   1:  PR[91,3] = PR[90,3] + 81.571;
   1:L PR[91] R[100]mm/sec CNT100;
   1:  PR[91,1] = PR[90,1] + 62.644;
   1:  PR[91,2] = PR[90,2] + 12.917;
   1:  PR[91,3] = PR[90,3] + 81.586;
   1:L PR[91] R[100]mm/sec CNT100;
   1:  PR[91,1] = PR[90,1] + 61.308;
   1:  PR[91,2] = PR[90,2] + 14.480;
   1:  PR[91,3] = PR[90,3] + 81.595;
   1:L PR[91] R[100]mm/sec CNT100;
   1:  PR[91,1] = PR[90,1] + 59.721;
   1:  PR[91,2] = PR[90,2] + 15.862;
   1:  PR[91,3] = PR[90,3] + 81.603;
   1:L PR[91] R[100]mm/sec CNT100;
   1:  PR[91,1] = PR[90,1] + 58.345;
   1:  PR[91,2] = PR[90,2] + 17.260;
   1:  PR[91,3] = PR[90,3] + 81.612;
   1:L PR[91] R[100]mm/sec CNT100;
   1:  PR[91,1] = PR[90,1] + 57.004;
   1:  PR[91,2] = PR[90,2] + 18.393;
   1:  PR[91,3] = PR[90,3] + 81.620;
   1:L PR[91] R[100]mm/sec CNT100;
   1:  PR[91,1] = PR[90,1] + 55.414;
   1:  PR[91,2] = PR[90,2] + 19.586;
   1:  PR[91,3] = PR[90,3] + 81.627;
   1:L PR[91] R[100]mm/sec CNT100;
   1:  PR[91,1] = PR[90,1] + 53.101;
   1:  PR[91,2] = PR[90,2] + 20.989;
   1:  PR[91,3] = PR[90,3] + 81.635;
   1:L PR[91] R[100]mm/sec CNT100;
   1:  PR[91,1] = PR[90,1] + 51.821;
   1:  PR[91,2] = PR[90,2] + 21.944;
   1:  PR[91,3] = PR[90,3] + 81.646;
   1:L PR[91] R[100]mm/sec CNT100;
   1:  PR[91,1] = PR[90,1] + 50.965;
   1:  PR[91,2] = PR[90,2] + 22.483;
   1:  PR[91,3] = PR[90,3] + 81.652;
   1:L PR[91] R[100]mm/sec CNT100;
   1:  PR[91,1] = PR[90,1] + 48.444;
   1:  PR[91,2] = PR[90,2] + 23.798;
   1:  PR[91,3] = PR[90,3] + 81.656;
   1:L PR[91] R[100]mm/sec CNT100;
   1:  PR[91,1] = PR[90,1] + 44.728;
   1:  PR[91,2] = PR[90,2] + 25.350;
   1:  PR[91,3] = PR[90,3] + 81.668;
   1:L PR[91] R[100]mm/sec CNT100;
   1:  PR[91,1] = PR[90,1] + 44.378;
   1:  PR[91,2] = PR[90,2] + 25.468;
   1:  PR[91,3] = PR[90,3] + 81.684;
   1:L PR[91] R[100]mm/sec CNT100;
   1:  PR[91,1] = PR[90,1] + 43.418;
   1:  PR[91,2] = PR[90,2] + 25.698;
   1:  PR[91,3] = PR[90,3] + 81.685;
   1:L PR[91] R[100]mm/sec CNT100;
   1:  PR[91,1] = PR[90,1] + 39.402;
   1:  PR[91,2] = PR[90,2] + 26.808;
   1:  PR[91,3] = PR[90,3] + 81.689;
   1:L PR[91] R[100]mm/sec CNT100;
   1:  PR[91,1] = PR[90,1] + 37.303;
   1:  PR[91,2] = PR[90,2] + 27.046;
   1:  PR[91,3] = PR[90,3] + 81.706;
   1:L PR[91] R[100]mm/sec CNT100;
   1:  PR[91,1] = PR[90,1] + 34.276;
   1:  PR[91,2] = PR[90,2] + 27.336;
   1:  PR[91,3] = PR[90,3] + 81.714;
   1:L PR[91] R[100]mm/sec CNT100;
   1:  PR[91,1] = PR[90,1] + 29.886;
   1:  PR[91,2] = PR[90,2] + 27.088;
   1:  PR[91,3] = PR[90,3] + 81.727;
   1:L PR[91] R[100]mm/sec CNT100;
   1:  PR[91,1] = PR[90,1] + 29.056;
   1:  PR[91,2] = PR[90,2] + 27.022;
   1:  PR[91,3] = PR[90,3] + 81.744;
   1:L PR[91] R[100]mm/sec CNT100;
   1:  PR[91,1] = PR[90,1] + 26.131;
   1:  PR[91,2] = PR[90,2] + 26.352;
   1:  PR[91,3] = PR[90,3] + 81.748;
   1:L PR[91] R[100]mm/sec CNT100;
   1:  PR[91,1] = PR[90,1] + 23.532;
   1:  PR[91,2] = PR[90,2] + 25.732;
   1:  PR[91,3] = PR[90,3] + 81.760;
   1:L PR[91] R[100]mm/sec CNT100;
   1:  PR[91,1] = PR[90,1] + 17.636;
   1:  PR[91,2] = PR[90,2] + 25.942;
   1:  PR[91,3] = PR[90,3] + 81.770;
   1:L PR[91] R[100]mm/sec CNT100;
   1:  PR[91,1] = PR[90,1] + 16.885;
   1:  PR[91,2] = PR[90,2] + 25.956;
   1:  PR[91,3] = PR[90,3] + 81.794;
   1:L PR[91] R[100]mm/sec CNT100;
   1:  PR[91,1] = PR[90,1] + 16.176;
   1:  PR[91,2] = PR[90,2] + 25.869;
   1:  PR[91,3] = PR[90,3] + 81.797;
   1:L PR[91] R[100]mm/sec CNT100;
   1:  PR[91,1] = PR[90,1] + 15.321;
   1:  PR[91,2] = PR[90,2] + 25.726;
   1:  PR[91,3] = PR[90,3] + 81.800;
   1:L PR[91] R[100]mm/sec CNT100;
   1:  PR[91,1] = PR[90,1] + 10.804;
   1:  PR[91,2] = PR[90,2] + 24.798;
   1:  PR[91,3] = PR[90,3] + 81.804;
   1:L PR[91] R[100]mm/sec CNT100;
   1:  PR[91,1] = PR[90,1] + 8.361;
   1:  PR[91,2] = PR[90,2] + 25.041;
   1:  PR[91,3] = PR[90,3] + 81.822;
   1:L PR[91] R[100]mm/sec CNT100;
   1:  PR[91,1] = PR[90,1] + 6.155;
   1:  PR[91,2] = PR[90,2] + 25.303;
   1:  PR[91,3] = PR[90,3] + 81.832;
   1:L PR[91] R[100]mm/sec CNT100;
   1:  PR[91,1] = PR[90,1] + 5.173;
   1:  PR[91,2] = PR[90,2] + 25.372;
   1:  PR[91,3] = PR[90,3] + 81.841;
   1:L PR[91] R[100]mm/sec CNT100;
   1:  PR[91,1] = PR[90,1] + 1.298;
   1:  PR[91,2] = PR[90,2] + 25.364;
   1:  PR[91,3] = PR[90,3] + 81.845;
   1:L PR[91] R[100]mm/sec CNT100;
   1:  PR[91,1] = PR[90,1] + -2.664;
   1:  PR[91,2] = PR[90,2] + 24.963;
   1:  PR[91,3] = PR[90,3] + 81.860;
   1:L PR[91] R[100]mm/sec CNT100;
   1:  PR[91,1] = PR[90,1] + -5.173;
   1:  PR[91,2] = PR[90,2] + 25.202;
   1:  PR[91,3] = PR[90,3] + 81.876;
   1:L PR[91] R[100]mm/sec CNT100;
   1:  PR[91,1] = PR[90,1] + -5.712;
   1:  PR[91,2] = PR[90,2] + 25.242;
   1:  PR[91,3] = PR[90,3] + 81.887;
   1:L PR[91] R[100]mm/sec CNT100;
   1:  PR[91,1] = PR[90,1] + -11.323;
   1:  PR[91,2] = PR[90,2] + 25.461;
   1:  PR[91,3] = PR[90,3] + 81.889;
   1:L PR[91] R[100]mm/sec CNT100;
   1:  PR[91,1] = PR[90,1] + -16.101;
   1:  PR[91,2] = PR[90,2] + 25.612;
   1:  PR[91,3] = PR[90,3] + 81.911;
   1:L PR[91] R[100]mm/sec CNT100;
   1:  PR[91,1] = PR[90,1] + -25.910;
   1:  PR[91,2] = PR[90,2] + 25.277;
   1:  PR[91,3] = PR[90,3] + 81.930;
   1:L PR[91] R[100]mm/sec CNT100;
   1:  PR[91,1] = PR[90,1] + -34.129;
   1:  PR[91,2] = PR[90,2] + 24.417;
   1:  PR[91,3] = PR[90,3] + 81.970;
   1:L PR[91] R[100]mm/sec CNT100;
   1:  PR[91,1] = PR[90,1] + -42.483;
   1:  PR[91,2] = PR[90,2] + 22.838;
   1:  PR[91,3] = PR[90,3] + 82.003;
   1:L PR[91] R[100]mm/sec CNT100;
   1:  PR[91,1] = PR[90,1] + -43.134;
   1:  PR[91,2] = PR[90,2] + 22.635;
   1:  PR[91,3] = PR[90,3] + 82.037;
   1:L PR[91] R[100]mm/sec CNT100;
   1:  PR[91,1] = PR[90,1] + -49.319;
   1:  PR[91,2] = PR[90,2] + 20.568;
   1:  PR[91,3] = PR[90,3] + 82.040;
   1:L PR[91] R[100]mm/sec CNT100;
   1:  PR[91,1] = PR[90,1] + -54.015;
   1:  PR[91,2] = PR[90,2] + 18.303;
   1:  PR[91,3] = PR[90,3] + 82.066;
   1:L PR[91] R[100]mm/sec CNT100;
   1:  PR[91,1] = PR[90,1] + -55.257;
   1:  PR[91,2] = PR[90,2] + 17.653;
   1:  PR[91,3] = PR[90,3] + 82.087;
   1:L PR[91] R[100]mm/sec CNT100;
   1:  PR[91,1] = PR[90,1] + -55.728;
   1:  PR[91,2] = PR[90,2] + 17.390;
   1:  PR[91,3] = PR[90,3] + 82.093;
   1:L PR[91] R[100]mm/sec CNT100;
   1:  PR[91] = PR[90];
   1:  PR[91,1] = PR[90,1] + -58.434;
   1:  PR[91,2] = PR[90,2] + 14.368;
   1:  PR[91,3] = PR[90,3] + 83.395;
   1:L PR[91] R[100]mm/sec CNT100;
   1:  PR[91,1] = PR[90,1] + -59.656;
   1:  PR[91,2] = PR[90,2] + 13.353;
   1:  PR[91,3] = PR[90,3] + 82.114;
   1:L PR[91] R[100]mm/sec CNT100;
   1:  PR[91,1] = PR[90,1] + -61.596;
   1:  PR[91,2] = PR[90,2] + 10.973;
   1:  PR[91,3] = PR[90,3] + 82.120;
   1:L PR[91] R[100]mm/sec CNT100;
   1:  PR[91,1] = PR[90,1] + -63.324;
   1:  PR[91,2] = PR[90,2] + 8.772;
   1:  PR[91,3] = PR[90,3] + 82.133;
   1:L PR[91] R[100]mm/sec CNT100;
   1:  PR[91,1] = PR[90,1] + -64.034;
   1:  PR[91,2] = PR[90,2] + 7.229;
   1:  PR[91,3] = PR[90,3] + 82.144;
   1:L PR[91] R[100]mm/sec CNT100;
   1:  PR[91,1] = PR[90,1] + -65.452;
   1:  PR[91,2] = PR[90,2] + 4.047;
   1:  PR[91,3] = PR[90,3] + 82.151;
   1:L PR[91] R[100]mm/sec CNT100;
   1:  PR[91,1] = PR[90,1] + -66.056;
   1:  PR[91,2] = PR[90,2] + -0.072;
   1:  PR[91,3] = PR[90,3] + 82.165;
   1:L PR[91] R[100]mm/sec CNT100;
   1:  PR[91,1] = PR[90,1] + -66.225;
   1:  PR[91,2] = PR[90,2] + -0.783;
   1:  PR[91,3] = PR[90,3] + 82.182;
   1:L PR[91] R[100]mm/sec CNT100;
   1:  PR[91,1] = PR[90,1] + -66.065;
   1:  PR[91,2] = PR[90,2] + -1.662;
   1:  PR[91,3] = PR[90,3] + 82.185;
   1:L PR[91] R[100]mm/sec CNT100;
   1:  PR[91,1] = PR[90,1] + -65.682;
   1:  PR[91,2] = PR[90,2] + -3.041;
   1:  PR[91,3] = PR[90,3] + 82.189;
   1:L PR[91] R[100]mm/sec CNT100;
   1:  PR[91,1] = PR[90,1] + -65.361;
   1:  PR[91,2] = PR[90,2] + -5.445;
   1:  PR[91,3] = PR[90,3] + 82.195;
   1:L PR[91] R[100]mm/sec CNT100;
   1:  PR[91,1] = PR[90,1] + -64.283;
   1:  PR[91,2] = PR[90,2] + -8.061;
   1:  PR[91,3] = PR[90,3] + 82.205;
   1:L PR[91] R[100]mm/sec CNT100;
   1:  PR[91,1] = PR[90,1] + -63.445;
   1:  PR[91,2] = PR[90,2] + -9.958;
   1:  PR[91,3] = PR[90,3] + 82.216;
   1:L PR[91] R[100]mm/sec CNT100;
   1:  PR[91,1] = PR[90,1] + -60.998;
   1:  PR[91,2] = PR[90,2] + -13.327;
   1:  PR[91,3] = PR[90,3] + 82.225;
   1:L PR[91] R[100]mm/sec CNT100;
   1:  PR[91,1] = PR[90,1] + -60.372;
   1:  PR[91,2] = PR[90,2] + -14.130;
   1:  PR[91,3] = PR[90,3] + 82.242;
   1:L PR[91] R[100]mm/sec CNT100;
   1:  PR[91,1] = PR[90,1] + -57.789;
   1:  PR[91,2] = PR[90,2] + -16.460;
   1:  PR[91,3] = PR[90,3] + 82.246;
   1:L PR[91] R[100]mm/sec CNT100;
   1:  PR[91,1] = PR[90,1] + -56.374;
   1:  PR[91,2] = PR[90,2] + -17.599;
   1:  PR[91,3] = PR[90,3] + 82.260;
   1:L PR[91] R[100]mm/sec CNT100;
   1:  PR[91,1] = PR[90,1] + -55.956;
   1:  PR[91,2] = PR[90,2] + -17.921;
   1:  PR[91,3] = PR[90,3] + 82.267;
   1:L PR[91] R[100]mm/sec CNT100;
   1:  PR[91,1] = PR[90,1] + -51.998;
   1:  PR[91,2] = PR[90,2] + -20.108;
   1:  PR[91,3] = PR[90,3] + 82.269;
   1:L PR[91] R[100]mm/sec CNT100;
   1:  PR[91,1] = PR[90,1] + -49.080;
   1:  PR[91,2] = PR[90,2] + -21.626;
   1:  PR[91,3] = PR[90,3] + 82.288;
   1:L PR[91] R[100]mm/sec CNT100;
   1:  PR[91,1] = PR[90,1] + -47.201;
   1:  PR[91,2] = PR[90,2] + -22.328;
   1:  PR[91,3] = PR[90,3] + 82.301;
   1:L PR[91] R[100]mm/sec CNT100;
   1:  PR[91,1] = PR[90,1] + -43.991;
   1:  PR[91,2] = PR[90,2] + -23.424;
   1:  PR[91,3] = PR[90,3] + 82.309;
   1:L PR[91] R[100]mm/sec CNT100;
   1:  PR[91,1] = PR[90,1] + -41.563;
   1:  PR[91,2] = PR[90,2] + -24.162;
   1:  PR[91,3] = PR[90,3] + 82.323;
   1:L PR[91] R[100]mm/sec CNT100;
   1:  PR[91,1] = PR[90,1] + -40.306;
   1:  PR[91,2] = PR[90,2] + -24.526;
   1:  PR[91,3] = PR[90,3] + 82.334;
   1:L PR[91] R[100]mm/sec CNT100;
   1:  PR[91,1] = PR[90,1] + -32.552;
   1:  PR[91,2] = PR[90,2] + -26.021;
   1:  PR[91,3] = PR[90,3] + 82.339;
   1:L PR[91] R[100]mm/sec CNT100;
   1:  PR[91,1] = PR[90,1] + -23.360;
   1:  PR[91,2] = PR[90,2] + -26.980;
   1:  PR[91,3] = PR[90,3] + 82.371;
   1:L PR[91] R[100]mm/sec CNT100;
   1:  PR[91,1] = PR[90,1] + -20.690;
   1:  PR[91,2] = PR[90,2] + -27.083;
   1:  PR[91,3] = PR[90,3] + 82.409;
   1:L PR[91] R[100]mm/sec CNT100;
   1:  PR[91,1] = PR[90,1] + -13.475;
   1:  PR[91,2] = PR[90,2] + -27.323;
   1:  PR[91,3] = PR[90,3] + 82.419;
   1:L PR[91] R[100]mm/sec CNT100;
   1:  PR[91,1] = PR[90,1] + -7.674;
   1:  PR[91,2] = PR[90,2] + -27.140;
   1:  PR[91,3] = PR[90,3] + 82.449;
   1:L PR[91] R[100]mm/sec CNT100;
   1:  PR[91,1] = PR[90,1] + -3.302;
   1:  PR[91,2] = PR[90,2] + -26.977;
   1:  PR[91,3] = PR[90,3] + 82.472;
   1:L PR[91] R[100]mm/sec CNT100;
   1:  PR[91,1] = PR[90,1] + -2.382;
   1:  PR[91,2] = PR[90,2] + -26.911;
   1:  PR[91,3] = PR[90,3] + 82.490;
   1:L PR[91] R[100]mm/sec CNT100;
   1:  PR[91,1] = PR[90,1] + -1.409;
   1:  PR[91,2] = PR[90,2] + -26.800;
   1:  PR[91,3] = PR[90,3] + 82.494;
   1:L PR[91] R[100]mm/sec CNT100;
   1:  PR[91,1] = PR[90,1] + -0.887;
   1:  PR[91,2] = PR[90,2] + -26.786;
   1:  PR[91,3] = PR[90,3] + 82.498;
   1:L PR[91] R[100]mm/sec CNT100;
   1:  PR[91,1] = PR[90,1] + 0.830;
   1:  PR[91,2] = PR[90,2] + -26.965;
   1:  PR[91,3] = PR[90,3] + 82.500;
   1:L PR[91] R[100]mm/sec CNT100;
   1:  PR[91,1] = PR[90,1] + 1.945;
   1:  PR[91,2] = PR[90,2] + -27.037;
   1:  PR[91,3] = PR[90,3] + 82.507;
   1:L PR[91] R[100]mm/sec CNT100;
   1:  PR[91,1] = PR[90,1] + 6.664;
   1:  PR[91,2] = PR[90,2] + -27.047;
   1:  PR[91,3] = PR[90,3] + 82.512;
   1:L PR[91] R[100]mm/sec CNT100;
   1:  PR[91,1] = PR[90,1] + 11.342;
   1:  PR[91,2] = PR[90,2] + -26.579;
   1:  PR[91,3] = PR[90,3] + 82.531;
   1:L PR[91] R[100]mm/sec CNT100;
   1:  PR[91,1] = PR[90,1] + 14.086;
   1:  PR[91,2] = PR[90,2] + -27.144;
   1:  PR[91,3] = PR[90,3] + 82.550;
   1:L PR[91] R[100]mm/sec CNT100;
   1:  PR[91,1] = PR[90,1] + 15.681;
   1:  PR[91,2] = PR[90,2] + -27.410;
   1:  PR[91,3] = PR[90,3] + 82.561;
   1:L PR[91] R[100]mm/sec CNT100;
   1:  PR[91,1] = PR[90,1] + 17.081;
   1:  PR[91,2] = PR[90,2] + -27.582;
   1:  PR[91,3] = PR[90,3] + 82.568;
   1:L PR[91] R[100]mm/sec CNT100;
   1:  PR[91,1] = PR[90,1] + 21.770;
   1:  PR[91,2] = PR[90,2] + -27.421;
   1:  PR[91,3] = PR[90,3] + 82.574;
   1:L PR[91] R[100]mm/sec CNT100;
   1:  PR[91,1] = PR[90,1] + 23.238;
   1:  PR[91,2] = PR[90,2] + -27.394;
   1:  PR[91,3] = PR[90,3] + 82.593;
   1:L PR[91] R[100]mm/sec CNT100;
   1:  PR[91,1] = PR[90,1] + 28.693;
   1:  PR[91,2] = PR[90,2] + -28.697;
   1:  PR[91,3] = PR[90,3] + 82.599;
   1:L PR[91] R[100]mm/sec CNT100;
   1:  PR[91,1] = PR[90,1] + 33.940;
   1:  PR[91,2] = PR[90,2] + -28.994;
   1:  PR[91,3] = PR[90,3] + 82.622;
   1:L PR[91] R[100]mm/sec CNT100;
   1:  PR[91,1] = PR[90,1] + 35.567;
   1:  PR[91,2] = PR[90,2] + -28.838;
   1:  PR[91,3] = PR[90,3] + 82.643;
   1:L PR[91] R[100]mm/sec CNT100;
   1:  PR[91,1] = PR[90,1] + 39.097;
   1:  PR[91,2] = PR[90,2] + -28.439;
   1:  PR[91,3] = PR[90,3] + 82.650;
   1:L PR[91] R[100]mm/sec CNT100;
   1:  PR[91,1] = PR[90,1] + 44.014;
   1:  PR[91,2] = PR[90,2] + -27.069;
   1:  PR[91,3] = PR[90,3] + 82.664;
   1:L PR[91] R[100]mm/sec CNT100;
   1:  PR[91,1] = PR[90,1] + 45.411;
   1:  PR[91,2] = PR[90,2] + -26.404;
   1:  PR[91,3] = PR[90,3] + 82.685;
   1:L PR[91] R[100]mm/sec CNT100;
   1:  PR[91,1] = PR[90,1] + 48.413;
   1:  PR[91,2] = PR[90,2] + -25.150;
   1:  PR[91,3] = PR[90,3] + 82.691;
   1:L PR[91] R[100]mm/sec CNT100;
   1:  PR[91,1] = PR[90,1] + 49.771;
   1:  PR[91,2] = PR[90,2] + -24.441;
   1:  PR[91,3] = PR[90,3] + 82.704;
   1:L PR[91] R[100]mm/sec CNT100;
   1:  PR[91,1] = PR[90,1] + 51.872;
   1:  PR[91,2] = PR[90,2] + -23.119;
   1:  PR[91,3] = PR[90,3] + 82.711;
   1:L PR[91] R[100]mm/sec CNT100;
   1:  PR[91,1] = PR[90,1] + 54.743;
   1:  PR[91,2] = PR[90,2] + -20.976;
   1:  PR[91,3] = PR[90,3] + 82.721;
   1:L PR[91] R[100]mm/sec CNT100;
   1:  PR[91,1] = PR[90,1] + 55.025;
   1:  PR[91,2] = PR[90,2] + -20.805;
   1:  PR[91,3] = PR[90,3] + 82.735;
   1:L PR[91] R[100]mm/sec CNT100;
   1:  PR[91,1] = PR[90,1] + 55.110;
   1:  PR[91,2] = PR[90,2] + -20.741;
   1:  PR[91,3] = PR[90,3] + 82.737;
   1:L PR[91] R[100]mm/sec CNT100;
   1:  PR[91,1] = PR[90,1] + 58.032;
   1:  PR[91,2] = PR[90,2] + -18.269;
   1:L PR[91] R[100]mm/sec CNT100;
   1:  PR[91,1] = PR[90,1] + 60.135;
   1:  PR[91,2] = PR[90,2] + -16.134;
   1:  PR[91,3] = PR[90,3] + 82.753;
   1:L PR[91] R[100]mm/sec CNT100;
   1:  PR[91,1] = PR[90,1] + 60.343;
   1:  PR[91,2] = PR[90,2] + -15.885;
   1:  PR[91,3] = PR[90,3] + 82.765;
   1:L PR[91] R[100]mm/sec CNT100;
   1:  PR[91,1] = PR[90,1] + 60.701;
   1:  PR[91,2] = PR[90,2] + -15.382;
   1:  PR[91,3] = PR[90,3] + 82.766;
   1:L PR[91] R[100]mm/sec CNT100;
   1:  PR[91,1] = PR[90,1] + 63.112;
   1:  PR[91,2] = PR[90,2] + -12.476;
   1:  PR[91,3] = PR[90,3] + 82.769;
   1:L PR[91] R[100]mm/sec CNT100;
   1:  PR[91,1] = PR[90,1] + 64.370;
   1:  PR[91,2] = PR[90,2] + -10.310;
   1:  PR[91,3] = PR[90,3] + 82.784;
   1:L PR[91] R[100]mm/sec CNT100;
   1:  PR[91,1] = PR[90,1] + 65.235;
   1:  PR[91,2] = PR[90,2] + -8.772;
   1:  PR[91,3] = PR[90,3] + 82.794;
   1:L PR[91] R[100]mm/sec CNT100;
   1:  PR[91,1] = PR[90,1] + 66.569;
   1:  PR[91,2] = PR[90,2] + -4.806;
   1:  PR[91,3] = PR[90,3] + 82.801;
   1:L PR[91] R[100]mm/sec CNT100;
   1:  PR[91,1] = PR[90,1] + 67.020;
   1:  PR[91,2] = PR[90,2] + -0.729;
   1:  PR[91,3] = PR[90,3] + 82.818;
   1:L PR[91] R[100]mm/sec CNT100;
   1:  PR[91,1] = PR[90,1] + 66.569;
   1:  PR[91,2] = PR[90,2] + 3.347;
   1:  PR[91,3] = PR[90,3] + 82.835;
   1:L PR[91] R[100]mm/sec CNT100;
   1:  PR[91,1] = PR[90,1] + 65.235;
   1:  PR[91,2] = PR[90,2] + 7.313;
   1:  PR[91,3] = PR[90,3] + 82.852;
   1:L PR[91] R[100]mm/sec CNT100;
   1:  PR[91,1] = PR[90,1] + 64.370;
   1:  PR[91,2] = PR[90,2] + 8.852;
   1:  PR[91,3] = PR[90,3] + 82.869;
   1:L PR[91] R[100]mm/sec CNT100;
   1:  PR[91,1] = PR[90,1] + 63.112;
   1:  PR[91,2] = PR[90,2] + 11.017;
   1:  PR[91,3] = PR[90,3] + 82.876;
   1:L PR[91] R[100]mm/sec CNT100;
   1:  PR[91,1] = PR[90,1] + 60.701;
   1:  PR[91,2] = PR[90,2] + 13.923;
   1:  PR[91,3] = PR[90,3] + 82.886;
   1:L PR[91] R[100]mm/sec CNT100;
   1:  PR[91,1] = PR[90,1] + 60.343;
   1:  PR[91,2] = PR[90,2] + 14.427;
   1:  PR[91,3] = PR[90,3] + 82.902;
   1:L PR[91] R[100]mm/sec CNT100;
   1:  PR[91,1] = PR[90,1] + 60.135;
   1:  PR[91,2] = PR[90,2] + 14.675;
   1:  PR[91,3] = PR[90,3] + 82.904;
   1:L PR[91] R[100]mm/sec CNT100;
   1:  PR[91,1] = PR[90,1] + 58.032;
   1:  PR[91,2] = PR[90,2] + 16.811;
   1:  PR[91,3] = PR[90,3] + 82.905;
   1:L PR[91] R[100]mm/sec CNT100;
   1:  PR[91,1] = PR[90,1] + 55.110;
   1:  PR[91,2] = PR[90,2] + 19.282;
   1:  PR[91,3] = PR[90,3] + 82.918;
   1:L PR[91] R[100]mm/sec CNT100;
   1:  PR[91,1] = PR[90,1] + 55.025;
   1:  PR[91,2] = PR[90,2] + 19.346;
   1:  PR[91,3] = PR[90,3] + 82.933;
   1:L PR[91] R[100]mm/sec CNT100;
   1:  PR[91,1] = PR[90,1] + 54.743;
   1:  PR[91,2] = PR[90,2] + 19.517;
   1:  PR[91,3] = PR[90,3] + 82.934;
   1:L PR[91] R[100]mm/sec CNT100;
   1:  PR[91,1] = PR[90,1] + 51.872;
   1:  PR[91,2] = PR[90,2] + 21.660;
   1:  PR[91,3] = PR[90,3] + 82.935;
   1:L PR[91] R[100]mm/sec CNT100;
   1:  PR[91,1] = PR[90,1] + 49.772;
   1:  PR[91,2] = PR[90,2] + 22.983;
   1:  PR[91,3] = PR[90,3] + 82.950;
   1:L PR[91] R[100]mm/sec CNT100;
   1:  PR[91,1] = PR[90,1] + 48.413;
   1:  PR[91,2] = PR[90,2] + 23.691;
   1:  PR[91,3] = PR[90,3] + 82.960;
   1:L PR[91] R[100]mm/sec CNT100;
   1:  PR[91,1] = PR[90,1] + 45.411;
   1:  PR[91,2] = PR[90,2] + 24.945;
   1:  PR[91,3] = PR[90,3] + 82.966;
   1:L PR[91] R[100]mm/sec CNT100;
   1:  PR[91,1] = PR[90,1] + 44.014;
   1:  PR[91,2] = PR[90,2] + 25.611;
   1:  PR[91,3] = PR[90,3] + 82.979;
   1:L PR[91] R[100]mm/sec CNT100;
   1:  PR[91,1] = PR[90,1] + 39.097;
   1:  PR[91,2] = PR[90,2] + 26.980;
   1:  PR[91,3] = PR[90,3] + 82.985;
   1:L PR[91] R[100]mm/sec CNT100;
   1:  PR[91,1] = PR[90,1] + 35.567;
   1:  PR[91,2] = PR[90,2] + 27.379;
   1:  PR[91,3] = PR[90,3] + 83.006;
   1:L PR[91] R[100]mm/sec CNT100;
   1:  PR[91,1] = PR[90,1] + 33.940;
   1:  PR[91,2] = PR[90,2] + 27.535;
   1:  PR[91,3] = PR[90,3] + 83.021;
   1:L PR[91] R[100]mm/sec CNT100;
   1:  PR[91,1] = PR[90,1] + 28.693;
   1:  PR[91,2] = PR[90,2] + 27.238;
   1:  PR[91,3] = PR[90,3] + 83.027;
   1:L PR[91] R[100]mm/sec CNT100;
   1:  PR[91,1] = PR[90,1] + 23.221;
   1:  PR[91,2] = PR[90,2] + 25.931;
   1:  PR[91,3] = PR[90,3] + 83.049;
   1:L PR[91] R[100]mm/sec CNT100;
   1:  PR[91,1] = PR[90,1] + 18.564;
   1:  PR[91,2] = PR[90,2] + 26.097;
   1:  PR[91,3] = PR[90,3] + 83.072;
   1:L PR[91] R[100]mm/sec CNT100;
   1:  PR[91,1] = PR[90,1] + 17.097;
   1:  PR[91,2] = PR[90,2] + 26.125;
   1:  PR[91,3] = PR[90,3] + 83.090;
   1:L PR[91] R[100]mm/sec CNT100;
   1:  PR[91,1] = PR[90,1] + 15.682;
   1:  PR[91,2] = PR[90,2] + 25.951;
   1:  PR[91,3] = PR[90,3] + 83.096;
   1:L PR[91] R[100]mm/sec CNT100;
   1:  PR[91,1] = PR[90,1] + 14.088;
   1:  PR[91,2] = PR[90,2] + 25.685;
   1:  PR[91,3] = PR[90,3] + 83.102;
   1:L PR[91] R[100]mm/sec CNT100;
   1:  PR[91,1] = PR[90,1] + 11.342;
   1:  PR[91,2] = PR[90,2] + 25.121;
   1:  PR[91,3] = PR[90,3] + 83.109;
   1:L PR[91] R[100]mm/sec CNT100;
   1:  PR[91,1] = PR[90,1] + 6.666;
   1:  PR[91,2] = PR[90,2] + 25.588;
   1:  PR[91,3] = PR[90,3] + 83.120;
   1:L PR[91] R[100]mm/sec CNT100;
   1:  PR[91,1] = PR[90,1] + 1.997;
   1:  PR[91,2] = PR[90,2] + 25.579;
   1:  PR[91,3] = PR[90,3] + 83.139;
   1:L PR[91] R[100]mm/sec CNT100;
   1:  PR[91,1] = PR[90,1] + -0.802;
   1:  PR[91,2] = PR[90,2] + 25.296;
   1:  PR[91,3] = PR[90,3] + 83.158;
   1:L PR[91] R[100]mm/sec CNT100;
   1:  PR[91,1] = PR[90,1] + -2.349;
   1:  PR[91,2] = PR[90,2] + 25.449;
   1:  PR[91,3] = PR[90,3] + 83.170;
   1:L PR[91] R[100]mm/sec CNT100;
   1:  PR[91,1] = PR[90,1] + -2.961;
   1:  PR[91,2] = PR[90,2] + 25.495;
   1:  PR[91,3] = PR[90,3] + 83.176;
   1:L PR[91] R[100]mm/sec CNT100;
   1:  PR[91,1] = PR[90,1] + -7.677;
   1:  PR[91,2] = PR[90,2] + 25.682;
   1:  PR[91,3] = PR[90,3] + 83.179;
   1:L PR[91] R[100]mm/sec CNT100;
   1:  PR[91,1] = PR[90,1] + -13.475;
   1:  PR[91,2] = PR[90,2] + 25.864;
   1:  PR[91,3] = PR[90,3] + 83.198;
   1:L PR[91] R[100]mm/sec CNT100;
   1:  PR[91,1] = PR[90,1] + -20.690;
   1:  PR[91,2] = PR[90,2] + 25.625;
   1:  PR[91,3] = PR[90,3] + 83.221;
   1:L PR[91] R[100]mm/sec CNT100;
   1:  PR[91,1] = PR[90,1] + -23.361;
   1:  PR[91,2] = PR[90,2] + 25.522;
   1:  PR[91,3] = PR[90,3] + 83.251;
   1:L PR[91] R[100]mm/sec CNT100;
   1:  PR[91,1] = PR[90,1] + -32.560;
   1:  PR[91,2] = PR[90,2] + 24.562;
   1:  PR[91,3] = PR[90,3] + 83.262;
   1:L PR[91] R[100]mm/sec CNT100;
   1:  PR[91,1] = PR[90,1] + -40.611;
   1:  PR[91,2] = PR[90,2] + 23.015;
   1:  PR[91,3] = PR[90,3] + 83.299;
   1:L PR[91] R[100]mm/sec CNT100;
   1:  PR[91,1] = PR[90,1] + -42.689;
   1:  PR[91,2] = PR[90,2] + 22.394;
   1:  PR[91,3] = PR[90,3] + 83.333;
   1:L PR[91] R[100]mm/sec CNT100;
   1:  PR[91,1] = PR[90,1] + -48.045;
   1:  PR[91,2] = PR[90,2] + 20.603;
   1:  PR[91,3] = PR[90,3] + 83.341;
   1:L PR[91] R[100]mm/sec CNT100;
   1:  PR[91,1] = PR[90,1] + -54.080;
   1:  PR[91,2] = PR[90,2] + 17.693;
   1:  PR[91,3] = PR[90,3] + 83.364;
   1:L PR[91] R[100]mm/sec CNT100;
   1:  PR[91,1] = PR[90,1] + -54.415;
   1:  PR[91,2] = PR[90,2] + 17.523;
   1:  PR[91,3] = PR[90,3] + 83.392;
   1:L PR[91] R[100]mm/sec CNT100;
   1:  PR[91,1] = PR[90,1] + -54.765;
   1:  PR[91,2] = PR[90,2] + 17.271;
   1:  PR[91,3] = PR[90,3] + 83.393;
   1:L PR[91] R[100]mm/sec CNT100;
   1:  PR[91] = PR[90];
   1:  PR[91,1] = PR[90,1] + -55.820;
   1:  PR[91,2] = PR[90,2] + 15.555;
   1:  PR[91,3] = PR[90,3] + 84.695;
   1:L PR[91] R[100]mm/sec CNT100;
   1:  PR[91,1] = PR[90,1] + -57.770;
   1:  PR[91,2] = PR[90,2] + 14.012;
   1:  PR[91,3] = PR[90,3] + 83.409;
   1:L PR[91] R[100]mm/sec CNT100;
   1:  PR[91,1] = PR[90,1] + -58.351;
   1:  PR[91,2] = PR[90,2] + 13.530;
   1:  PR[91,3] = PR[90,3] + 83.419;
   1:L PR[91] R[100]mm/sec CNT100;
   1:  PR[91,1] = PR[90,1] + -60.832;
   1:  PR[91,2] = PR[90,2] + 10.486;
   1:  PR[91,3] = PR[90,3] + 83.422;
   1:L PR[91] R[100]mm/sec CNT100;
   1:  PR[91,1] = PR[90,1] + -62.083;
   1:  PR[91,2] = PR[90,2] + 8.894;
   1:  PR[91,3] = PR[90,3] + 83.438;
   1:L PR[91] R[100]mm/sec CNT100;
   1:  PR[91,1] = PR[90,1] + -63.133;
   1:  PR[91,2] = PR[90,2] + 6.610;
   1:  PR[91,3] = PR[90,3] + 83.447;
   1:L PR[91] R[100]mm/sec CNT100;
   1:  PR[91,1] = PR[90,1] + -64.247;
   1:  PR[91,2] = PR[90,2] + 4.109;
   1:  PR[91,3] = PR[90,3] + 83.457;
   1:L PR[91] R[100]mm/sec CNT100;
   1:  PR[91,1] = PR[90,1] + -64.727;
   1:  PR[91,2] = PR[90,2] + 0.842;
   1:  PR[91,3] = PR[90,3] + 83.468;
   1:L PR[91] R[100]mm/sec CNT100;
   1:  PR[91,1] = PR[90,1] + -65.104;
   1:  PR[91,2] = PR[90,2] + -0.756;
   1:  PR[91,3] = PR[90,3] + 83.482;
   1:L PR[91] R[100]mm/sec CNT100;
   1:  PR[91,1] = PR[90,1] + -64.656;
   1:  PR[91,2] = PR[90,2] + -2.368;
   1:  PR[91,3] = PR[90,3] + 83.489;
   1:L PR[91] R[100]mm/sec CNT100;
   1:  PR[91,1] = PR[90,1] + -64.248;
   1:  PR[91,2] = PR[90,2] + -5.434;
   1:  PR[91,3] = PR[90,3] + 83.496;
   1:L PR[91] R[100]mm/sec CNT100;
   1:  PR[91,1] = PR[90,1] + -62.858;
   1:  PR[91,2] = PR[90,2] + -8.805;
   1:  PR[91,3] = PR[90,3] + 83.508;
   1:L PR[91] R[100]mm/sec CNT100;
   1:  PR[91,1] = PR[90,1] + -62.357;
   1:  PR[91,2] = PR[90,2] + -9.939;
   1:  PR[91,3] = PR[90,3] + 83.523;
   1:L PR[91] R[100]mm/sec CNT100;
   1:  PR[91,1] = PR[90,1] + -59.299;
   1:  PR[91,2] = PR[90,2] + -14.135;
   1:  PR[91,3] = PR[90,3] + 83.529;
   1:L PR[91] R[100]mm/sec CNT100;
   1:  PR[91,1] = PR[90,1] + -58.899;
   1:  PR[91,2] = PR[90,2] + -14.496;
   1:  PR[91,3] = PR[90,3] + 83.550;
   1:L PR[91] R[100]mm/sec CNT100;
   1:  PR[91,1] = PR[90,1] + -55.480;
   1:  PR[91,2] = PR[90,2] + -17.247;
   1:  PR[91,3] = PR[90,3] + 83.552;
   1:L PR[91] R[100]mm/sec CNT100;
   1:  PR[91,1] = PR[90,1] + -54.310;
   1:  PR[91,2] = PR[90,2] + -18.147;
   1:  PR[91,3] = PR[90,3] + 83.570;
   1:L PR[91] R[100]mm/sec CNT100;
   1:  PR[91,1] = PR[90,1] + -51.181;
   1:  PR[91,2] = PR[90,2] + -19.877;
   1:  PR[91,3] = PR[90,3] + 83.576;
   1:L PR[91] R[100]mm/sec CNT100;
   1:  PR[91,1] = PR[90,1] + -47.305;
   1:  PR[91,2] = PR[90,2] + -21.893;
   1:  PR[91,3] = PR[90,3] + 83.591;
   1:L PR[91] R[100]mm/sec CNT100;
   1:  PR[91,1] = PR[90,1] + -46.433;
   1:  PR[91,2] = PR[90,2] + -22.219;
   1:  PR[91,3] = PR[90,3] + 83.609;
   1:L PR[91] R[100]mm/sec CNT100;
   1:  PR[91,1] = PR[90,1] + -44.851;
   1:  PR[91,2] = PR[90,2] + -22.759;
   1:  PR[91,3] = PR[90,3] + 83.613;
   1:L PR[91] R[100]mm/sec CNT100;
   1:  PR[91,1] = PR[90,1] + -40.571;
   1:  PR[91,2] = PR[90,2] + -24.060;
   1:  PR[91,3] = PR[90,3] + 83.620;
   1:L PR[91] R[100]mm/sec CNT100;
   1:  PR[91,1] = PR[90,1] + -38.296;
   1:  PR[91,2] = PR[90,2] + -24.719;
   1:  PR[91,3] = PR[90,3] + 83.638;
   1:L PR[91] R[100]mm/sec CNT100;
   1:  PR[91,1] = PR[90,1] + -32.592;
   1:  PR[91,2] = PR[90,2] + -25.826;
   1:  PR[91,3] = PR[90,3] + 83.648;
   1:L PR[91] R[100]mm/sec CNT100;
   1:  PR[91,1] = PR[90,1] + -30.326;
   1:  PR[91,2] = PR[90,2] + -26.230;
   1:  PR[91,3] = PR[90,3] + 83.672;
   1:L PR[91] R[100]mm/sec CNT100;
   1:  PR[91,1] = PR[90,1] + -20.814;
   1:  PR[91,2] = PR[90,2] + -27.225;
   1:  PR[91,3] = PR[90,3] + 83.681;
   1:L PR[91] R[100]mm/sec CNT100;
   1:  PR[91,1] = PR[90,1] + -17.150;
   1:  PR[91,2] = PR[90,2] + -27.366;
   1:  PR[91,3] = PR[90,3] + 83.721;
   1:L PR[91] R[100]mm/sec CNT100;
   1:  PR[91,1] = PR[90,1] + -10.849;
   1:  PR[91,2] = PR[90,2] + -27.576;
   1:  PR[91,3] = PR[90,3] + 83.736;
   1:L PR[91] R[100]mm/sec CNT100;
   1:  PR[91,1] = PR[90,1] + -4.026;
   1:  PR[91,2] = PR[90,2] + -27.361;
   1:  PR[91,3] = PR[90,3] + 83.762;
   1:L PR[91] R[100]mm/sec CNT100;
   1:  PR[91,1] = PR[90,1] + -0.594;
   1:  PR[91,2] = PR[90,2] + -27.232;
   1:  PR[91,3] = PR[90,3] + 83.790;
   1:L PR[91] R[100]mm/sec CNT100;
   1:  PR[91,1] = PR[90,1] + 0.853;
   1:  PR[91,2] = PR[90,2] + -27.123;
   1:  PR[91,3] = PR[90,3] + 83.804;
   1:L PR[91] R[100]mm/sec CNT100;
   1:  PR[91,1] = PR[90,1] + 2.653;
   1:  PR[91,2] = PR[90,2] + -27.252;
   1:  PR[91,3] = PR[90,3] + 83.810;
   1:L PR[91] R[100]mm/sec CNT100;
   1:  PR[91,1] = PR[90,1] + 5.506;
   1:  PR[91,2] = PR[90,2] + -27.258;
   1:  PR[91,3] = PR[90,3] + 83.818;
   1:L PR[91] R[100]mm/sec CNT100;
   1:  PR[91,1] = PR[90,1] + 7.419;
   1:  PR[91,2] = PR[90,2] + -27.285;
   1:  PR[91,3] = PR[90,3] + 83.829;
   1:L PR[91] R[100]mm/sec CNT100;
   1:  PR[91,1] = PR[90,1] + 7.750;
   1:  PR[91,2] = PR[90,2] + -27.279;
   1:  PR[91,3] = PR[90,3] + 83.837;
   1:L PR[91] R[100]mm/sec CNT100;
   1:  PR[91,1] = PR[90,1] + 8.440;
   1:  PR[91,2] = PR[90,2] + -27.232;
   1:  PR[91,3] = PR[90,3] + 83.839;
   1:L PR[91] R[100]mm/sec CNT100;
   1:  PR[91,1] = PR[90,1] + 11.886;
   1:  PR[91,2] = PR[90,2] + -26.903;
   1:  PR[91,3] = PR[90,3] + 83.841;
   1:L PR[91] R[100]mm/sec CNT100;
   1:  PR[91,1] = PR[90,1] + 12.853;
   1:  PR[91,2] = PR[90,2] + -27.102;
   1:  PR[91,3] = PR[90,3] + 83.856;
   1:L PR[91] R[100]mm/sec CNT100;
   1:  PR[91,1] = PR[90,1] + 15.186;
   1:  PR[91,2] = PR[90,2] + -27.492;
   1:  PR[91,3] = PR[90,3] + 83.860;
   1:L PR[91] R[100]mm/sec CNT100;
   1:  PR[91,1] = PR[90,1] + 17.292;
   1:  PR[91,2] = PR[90,2] + -27.750;
   1:  PR[91,3] = PR[90,3] + 83.870;
   1:L PR[91] R[100]mm/sec CNT100;
   1:  PR[91,1] = PR[90,1] + 20.645;
   1:  PR[91,2] = PR[90,2] + -27.636;
   1:  PR[91,3] = PR[90,3] + 83.878;
   1:L PR[91] R[100]mm/sec CNT100;
   1:  PR[91,1] = PR[90,1] + 22.928;
   1:  PR[91,2] = PR[90,2] + -27.593;
   1:  PR[91,3] = PR[90,3] + 83.892;
   1:L PR[91] R[100]mm/sec CNT100;
   1:  PR[91,1] = PR[90,1] + 26.835;
   1:  PR[91,2] = PR[90,2] + -28.529;
   1:  PR[91,3] = PR[90,3] + 83.901;
   1:L PR[91] R[100]mm/sec CNT100;
   1:  PR[91,1] = PR[90,1] + 28.431;
   1:  PR[91,2] = PR[90,2] + -28.891;
   1:  PR[91,3] = PR[90,3] + 83.918;
   1:L PR[91] R[100]mm/sec CNT100;
   1:  PR[91,1] = PR[90,1] + 33.590;
   1:  PR[91,2] = PR[90,2] + -29.193;
   1:  PR[91,3] = PR[90,3] + 83.925;
   1:L PR[91] R[100]mm/sec CNT100;
   1:  PR[91,1] = PR[90,1] + 38.798;
   1:  PR[91,2] = PR[90,2] + -28.611;
   1:  PR[91,3] = PR[90,3] + 83.946;
   1:L PR[91] R[100]mm/sec CNT100;
   1:  PR[91,1] = PR[90,1] + 41.367;
   1:  PR[91,2] = PR[90,2] + -27.900;
   1:  PR[91,3] = PR[90,3] + 83.968;
   1:L PR[91] R[100]mm/sec CNT100;
   1:  PR[91,1] = PR[90,1] + 43.735;
   1:  PR[91,2] = PR[90,2] + -27.217;
   1:  PR[91,3] = PR[90,3] + 83.979;
   1:L PR[91] R[100]mm/sec CNT100;
   1:  PR[91,1] = PR[90,1] + 47.721;
   1:  PR[91,2] = PR[90,2] + -25.319;
   1:  PR[91,3] = PR[90,3] + 83.989;
   1:L PR[91] R[100]mm/sec CNT100;
   1:  PR[91,1] = PR[90,1] + 48.381;
   1:  PR[91,2] = PR[90,2] + -25.044;
   1:  PR[91,3] = PR[90,3] + 84.007;
   1:L PR[91] R[100]mm/sec CNT100;
   1:  PR[91,1] = PR[90,1] + 48.578;
   1:  PR[91,2] = PR[90,2] + -24.941;
   1:  PR[91,3] = PR[90,3] + 84.010;
   1:L PR[91] R[100]mm/sec CNT100;
   1:  PR[91,1] = PR[90,1] + 51.923;
   1:  PR[91,2] = PR[90,2] + -22.835;
   1:  PR[91,3] = PR[90,3] + 84.011;
   1:L PR[91] R[100]mm/sec CNT100;
   1:  PR[91,1] = PR[90,1] + 53.939;
   1:  PR[91,2] = PR[90,2] + -21.330;
   1:  PR[91,3] = PR[90,3] + 84.027;
   1:L PR[91] R[100]mm/sec CNT100;
   1:  PR[91,1] = PR[90,1] + 54.792;
   1:  PR[91,2] = PR[90,2] + -20.561;
   1:  PR[91,3] = PR[90,3] + 84.037;
   1:L PR[91] R[100]mm/sec CNT100;
   1:  PR[91,1] = PR[90,1] + 56.133;
   1:  PR[91,2] = PR[90,2] + -19.163;
   1:  PR[91,3] = PR[90,3] + 84.042;
   1:L PR[91] R[100]mm/sec CNT100;
   1:  PR[91,1] = PR[90,1] + 57.720;
   1:  PR[91,2] = PR[90,2] + -17.820;
   1:  PR[91,3] = PR[90,3] + 84.050;
   1:L PR[91] R[100]mm/sec CNT100;
   1:  PR[91,1] = PR[90,1] + 58.592;
   1:  PR[91,2] = PR[90,2] + -16.934;
   1:  PR[91,3] = PR[90,3] + 84.059;
   1:L PR[91] R[100]mm/sec CNT100;
   1:  PR[91,1] = PR[90,1] + 60.063;
   1:  PR[91,2] = PR[90,2] + -15.177;
   1:  PR[91,3] = PR[90,3] + 84.064;
   1:L PR[91] R[100]mm/sec CNT100;
   1:  PR[91,1] = PR[90,1] + 61.896;
   1:  PR[91,2] = PR[90,2] + -12.606;
   1:  PR[91,3] = PR[90,3] + 84.073;
   1:L PR[91] R[100]mm/sec CNT100;
   1:  PR[91,1] = PR[90,1] + 62.073;
   1:  PR[91,2] = PR[90,2] + -12.393;
   1:  PR[91,3] = PR[90,3] + 84.086;
   1:L PR[91] R[100]mm/sec CNT100;
   1:  PR[91,1] = PR[90,1] + 62.111;
   1:  PR[91,2] = PR[90,2] + -12.327;
   1:  PR[91,3] = PR[90,3] + 84.087;
   1:L PR[91] R[100]mm/sec CNT100;
   1:  PR[91,1] = PR[90,1] + 64.147;
   1:  PR[91,2] = PR[90,2] + -8.707;
   1:  PR[91,3] = PR[90,3] + 84.088;
   1:L PR[91] R[100]mm/sec CNT100;
   1:  PR[91,1] = PR[90,1] + 64.790;
   1:  PR[91,2] = PR[90,2] + -6.800;
   1:  PR[91,3] = PR[90,3] + 84.105;
   1:L PR[91] R[100]mm/sec CNT100;
   1:  PR[91,1] = PR[90,1] + 65.448;
   1:  PR[91,2] = PR[90,2] + -4.780;
   1:  PR[91,3] = PR[90,3] + 84.113;
   1:L PR[91] R[100]mm/sec CNT100;
   1:  PR[91,1] = PR[90,1] + 65.893;
   1:  PR[91,2] = PR[90,2] + -0.729;
   1:  PR[91,3] = PR[90,3] + 84.122;
   1:L PR[91] R[100]mm/sec CNT100;
   1:  PR[91,1] = PR[90,1] + 65.448;
   1:  PR[91,2] = PR[90,2] + 3.322;
   1:  PR[91,3] = PR[90,3] + 84.139;
   1:L PR[91] R[100]mm/sec CNT100;
   1:  PR[91,1] = PR[90,1] + 64.790;
   1:  PR[91,2] = PR[90,2] + 5.341;
   1:  PR[91,3] = PR[90,3] + 84.156;
   1:L PR[91] R[100]mm/sec CNT100;
   1:  PR[91,1] = PR[90,1] + 64.147;
   1:  PR[91,2] = PR[90,2] + 7.247;
   1:  PR[91,3] = PR[90,3] + 84.164;
   1:L PR[91] R[100]mm/sec CNT100;
   1:  PR[91,1] = PR[90,1] + 62.065;
   1:  PR[91,2] = PR[90,2] + 10.944;
   1:  PR[91,3] = PR[90,3] + 84.173;
   1:L PR[91] R[100]mm/sec CNT100;
   1:  PR[91,1] = PR[90,1] + 61.896;
   1:  PR[91,2] = PR[90,2] + 11.147;
   1:  PR[91,3] = PR[90,3] + 84.190;
   1:L PR[91] R[100]mm/sec CNT100;
   1:  PR[91,1] = PR[90,1] + 60.063;
   1:  PR[91,2] = PR[90,2] + 13.718;
   1:  PR[91,3] = PR[90,3] + 84.191;
   1:L PR[91] R[100]mm/sec CNT100;
   1:  PR[91,1] = PR[90,1] + 58.592;
   1:  PR[91,2] = PR[90,2] + 15.476;
   1:  PR[91,3] = PR[90,3] + 84.204;
   1:L PR[91] R[100]mm/sec CNT100;
   1:  PR[91,1] = PR[90,1] + 57.720;
   1:  PR[91,2] = PR[90,2] + 16.362;
   1:  PR[91,3] = PR[90,3] + 84.214;
   1:L PR[91] R[100]mm/sec CNT100;
   1:  PR[91,1] = PR[90,1] + 56.133;
   1:  PR[91,2] = PR[90,2] + 17.704;
   1:  PR[91,3] = PR[90,3] + 84.219;
   1:L PR[91] R[100]mm/sec CNT100;
   1:  PR[91,1] = PR[90,1] + 54.792;
   1:  PR[91,2] = PR[90,2] + 19.102;
   1:  PR[91,3] = PR[90,3] + 84.227;
   1:L PR[91] R[100]mm/sec CNT100;
   1:  PR[91,1] = PR[90,1] + 53.939;
   1:  PR[91,2] = PR[90,2] + 19.872;
   1:  PR[91,3] = PR[90,3] + 84.235;
   1:L PR[91] R[100]mm/sec CNT100;
   1:  PR[91,1] = PR[90,1] + 51.923;
   1:  PR[91,2] = PR[90,2] + 21.376;
   1:  PR[91,3] = PR[90,3] + 84.240;
   1:L PR[91] R[100]mm/sec CNT100;
   1:  PR[91,1] = PR[90,1] + 48.578;
   1:  PR[91,2] = PR[90,2] + 23.482;
   1:  PR[91,3] = PR[90,3] + 84.250;
   1:L PR[91] R[100]mm/sec CNT100;
   1:  PR[91,1] = PR[90,1] + 48.381;
   1:  PR[91,2] = PR[90,2] + 23.585;
   1:  PR[91,3] = PR[90,3] + 84.267;
   1:L PR[91] R[100]mm/sec CNT100;
   1:  PR[91,1] = PR[90,1] + 47.721;
   1:  PR[91,2] = PR[90,2] + 23.860;
   1:  PR[91,3] = PR[90,3] + 84.268;
   1:L PR[91] R[100]mm/sec CNT100;
   1:  PR[91,1] = PR[90,1] + 43.735;
   1:  PR[91,2] = PR[90,2] + 25.759;
   1:  PR[91,3] = PR[90,3] + 84.270;
   1:L PR[91] R[100]mm/sec CNT100;
   1:  PR[91,1] = PR[90,1] + 41.367;
   1:  PR[91,2] = PR[90,2] + 26.441;
   1:  PR[91,3] = PR[90,3] + 84.289;
   1:L PR[91] R[100]mm/sec CNT100;
   1:  PR[91,1] = PR[90,1] + 38.798;
   1:  PR[91,2] = PR[90,2] + 27.152;
   1:  PR[91,3] = PR[90,3] + 84.299;
   1:L PR[91] R[100]mm/sec CNT100;
   1:  PR[91,1] = PR[90,1] + 33.590;
   1:  PR[91,2] = PR[90,2] + 27.734;
   1:  PR[91,3] = PR[90,3] + 84.310;
   1:L PR[91] R[100]mm/sec CNT100;
   1:  PR[91,1] = PR[90,1] + 28.431;
   1:  PR[91,2] = PR[90,2] + 27.432;
   1:  PR[91,3] = PR[90,3] + 84.331;
   1:L PR[91] R[100]mm/sec CNT100;
   1:  PR[91,1] = PR[90,1] + 26.835;
   1:  PR[91,2] = PR[90,2] + 27.070;
   1:  PR[91,3] = PR[90,3] + 84.353;
   1:L PR[91] R[100]mm/sec CNT100;
   1:  PR[91,1] = PR[90,1] + 22.911;
   1:  PR[91,2] = PR[90,2] + 26.131;
   1:  PR[91,3] = PR[90,3] + 84.359;
   1:L PR[91] R[100]mm/sec CNT100;
   1:  PR[91,1] = PR[90,1] + 19.492;
   1:  PR[91,2] = PR[90,2] + 26.252;
   1:  PR[91,3] = PR[90,3] + 84.376;
   1:L PR[91] R[100]mm/sec CNT100;
   1:  PR[91,1] = PR[90,1] + 17.308;
   1:  PR[91,2] = PR[90,2] + 26.293;
   1:  PR[91,3] = PR[90,3] + 84.390;
   1:L PR[91] R[100]mm/sec CNT100;
   1:  PR[91,1] = PR[90,1] + 15.188;
   1:  PR[91,2] = PR[90,2] + 26.034;
   1:  PR[91,3] = PR[90,3] + 84.399;
   1:L PR[91] R[100]mm/sec CNT100;
   1:  PR[91,1] = PR[90,1] + 12.855;
   1:  PR[91,2] = PR[90,2] + 25.644;
   1:  PR[91,3] = PR[90,3] + 84.408;
   1:L PR[91] R[100]mm/sec CNT100;
   1:  PR[91,1] = PR[90,1] + 11.886;
   1:  PR[91,2] = PR[90,2] + 25.445;
   1:  PR[91,3] = PR[90,3] + 84.418;
   1:L PR[91] R[100]mm/sec CNT100;
   1:  PR[91,1] = PR[90,1] + 8.440;
   1:  PR[91,2] = PR[90,2] + 25.773;
   1:  PR[91,3] = PR[90,3] + 84.422;
   1:L PR[91] R[100]mm/sec CNT100;
   1:  PR[91,1] = PR[90,1] + 7.775;
   1:  PR[91,2] = PR[90,2] + 25.818;
   1:  PR[91,3] = PR[90,3] + 84.436;
   1:L PR[91] R[100]mm/sec CNT100;
   1:  PR[91,1] = PR[90,1] + 2.699;
   1:  PR[91,2] = PR[90,2] + 25.794;
   1:  PR[91,3] = PR[90,3] + 84.439;
   1:L PR[91] R[100]mm/sec CNT100;
   1:  PR[91,1] = PR[90,1] + 1.042;
   1:  PR[91,2] = PR[90,2] + 25.626;
   1:  PR[91,3] = PR[90,3] + 84.460;
   1:L PR[91] R[100]mm/sec CNT100;
   1:  PR[91,1] = PR[90,1] + 0.458;
   1:  PR[91,2] = PR[90,2] + 25.698;
   1:  PR[91,3] = PR[90,3] + 84.467;
   1:L PR[91] R[100]mm/sec CNT100;
   1:  PR[91,1] = PR[90,1] + -0.211;
   1:  PR[91,2] = PR[90,2] + 25.747;
   1:  PR[91,3] = PR[90,3] + 84.469;
   1:L PR[91] R[100]mm/sec CNT100;
   1:  PR[91,1] = PR[90,1] + -4.029;
   1:  PR[91,2] = PR[90,2] + 25.902;
   1:  PR[91,3] = PR[90,3] + 84.472;
   1:L PR[91] R[100]mm/sec CNT100;
   1:  PR[91,1] = PR[90,1] + -10.849;
   1:  PR[91,2] = PR[90,2] + 26.117;
   1:  PR[91,3] = PR[90,3] + 84.487;
   1:L PR[91] R[100]mm/sec CNT100;
   1:  PR[91,1] = PR[90,1] + -17.150;
   1:  PR[91,2] = PR[90,2] + 25.907;
   1:  PR[91,3] = PR[90,3] + 84.516;
   1:L PR[91] R[100]mm/sec CNT100;
   1:  PR[91,1] = PR[90,1] + -20.814;
   1:  PR[91,2] = PR[90,2] + 25.766;
   1:  PR[91,3] = PR[90,3] + 84.542;
   1:L PR[91] R[100]mm/sec CNT100;
   1:  PR[91,1] = PR[90,1] + -30.326;
   1:  PR[91,2] = PR[90,2] + 24.771;
   1:  PR[91,3] = PR[90,3] + 84.557;
   1:L PR[91] R[100]mm/sec CNT100;
   1:  PR[91,1] = PR[90,1] + -32.592;
   1:  PR[91,2] = PR[90,2] + 24.367;
   1:  PR[91,3] = PR[90,3] + 84.596;
   1:L PR[91] R[100]mm/sec CNT100;
   1:  PR[91,1] = PR[90,1] + -38.503;
   1:  PR[91,2] = PR[90,2] + 23.224;
   1:  PR[91,3] = PR[90,3] + 84.606;
   1:L PR[91] R[100]mm/sec CNT100;
   1:  PR[91,1] = PR[90,1] + -43.527;
   1:  PR[91,2] = PR[90,2] + 21.723;
   1:  PR[91,3] = PR[90,3] + 84.630;
   1:L PR[91] R[100]mm/sec CNT100;
   1:  PR[91,1] = PR[90,1] + -46.770;
   1:  PR[91,2] = PR[90,2] + 20.639;
   1:  PR[91,3] = PR[90,3] + 84.652;
   1:L PR[91] R[100]mm/sec CNT100;
   1:  PR[91,1] = PR[90,1] + -50.439;
   1:  PR[91,2] = PR[90,2] + 18.870;
   1:  PR[91,3] = PR[90,3] + 84.666;
   1:L PR[91] R[100]mm/sec CNT100;
   1:  PR[91,1] = PR[90,1] + -53.072;
   1:  PR[91,2] = PR[90,2] + 17.528;
   1:  PR[91,3] = PR[90,3] + 84.683;
   1:L PR[91] R[100]mm/sec CNT100;
   1:  PR[91] = PR[90];
   1:  PR[91,1] = PR[90,1] + -56.871;
   1:  PR[91,2] = PR[90,2] + 13.843;
   1:  PR[91,3] = PR[90,3] + 85.995;
   1:L PR[91] R[100]mm/sec CNT100;
   1:  PR[91,1] = PR[90,1] + -57.057;
   1:  PR[91,2] = PR[90,2] + 13.694;
   1:  PR[91,3] = PR[90,3] + 84.721;
   1:L PR[91] R[100]mm/sec CNT100;
   1:  PR[91,1] = PR[90,1] + -60.068;
   1:  PR[91,2] = PR[90,2] + 10.000;
   1:  PR[91,3] = PR[90,3] + 84.722;
   1:L PR[91] R[100]mm/sec CNT100;
   1:  PR[91,1] = PR[90,1] + -60.841;
   1:  PR[91,2] = PR[90,2] + 9.015;
   1:  PR[91,3] = PR[90,3] + 84.742;
   1:L PR[91] R[100]mm/sec CNT100;
   1:  PR[91,1] = PR[90,1] + -62.232;
   1:  PR[91,2] = PR[90,2] + 5.989;
   1:  PR[91,3] = PR[90,3] + 84.747;
   1:L PR[91] R[100]mm/sec CNT100;
   1:  PR[91,1] = PR[90,1] + -63.043;
   1:  PR[91,2] = PR[90,2] + 4.170;
   1:  PR[91,3] = PR[90,3] + 84.761;
   1:L PR[91] R[100]mm/sec CNT100;
   1:  PR[91,1] = PR[90,1] + -63.397;
   1:  PR[91,2] = PR[90,2] + 1.755;
   1:  PR[91,3] = PR[90,3] + 84.770;
   1:L PR[91] R[100]mm/sec CNT100;
   1:  PR[91,1] = PR[90,1] + -63.845;
   1:  PR[91,2] = PR[90,2] + -0.138;
   1:  PR[91,3] = PR[90,3] + 84.780;
   1:L PR[91] R[100]mm/sec CNT100;
   1:  PR[91,1] = PR[90,1] + -63.928;
   1:  PR[91,2] = PR[90,2] + -0.626;
   1:  PR[91,3] = PR[90,3] + 84.788;
   1:L PR[91] R[100]mm/sec CNT100;
   1:  PR[91,1] = PR[90,1] + -63.631;
   1:  PR[91,2] = PR[90,2] + -1.695;
   1:  PR[91,3] = PR[90,3] + 84.790;
   1:L PR[91] R[100]mm/sec CNT100;
   1:  PR[91,1] = PR[90,1] + -63.134;
   1:  PR[91,2] = PR[90,2] + -5.424;
   1:  PR[91,3] = PR[90,3] + 84.795;
   1:L PR[91] R[100]mm/sec CNT100;
   1:  PR[91,1] = PR[90,1] + -61.433;
   1:  PR[91,2] = PR[90,2] + -9.549;
   1:  PR[91,3] = PR[90,3] + 84.810;
   1:L PR[91] R[100]mm/sec CNT100;
   1:  PR[91,1] = PR[90,1] + -61.268;
   1:  PR[91,2] = PR[90,2] + -9.923;
   1:  PR[91,3] = PR[90,3] + 84.829;
   1:L PR[91] R[100]mm/sec CNT100;
   1:  PR[91,1] = PR[90,1] + -59.724;
   1:  PR[91,2] = PR[90,2] + -12.049;
   1:  PR[91,3] = PR[90,3] + 84.831;
   1:L PR[91] R[100]mm/sec CNT100;
   1:  PR[91,1] = PR[90,1] + -57.969;
   1:  PR[91,2] = PR[90,2] + -14.174;
   1:  PR[91,3] = PR[90,3] + 84.842;
   1:L PR[91] R[100]mm/sec CNT100;
   1:  PR[91,1] = PR[90,1] + -54.587;
   1:  PR[91,2] = PR[90,2] + -16.895;
   1:  PR[91,3] = PR[90,3] + 84.853;
   1:L PR[91] R[100]mm/sec CNT100;
   1:  PR[91,1] = PR[90,1] + -52.665;
   1:  PR[91,2] = PR[90,2] + -18.373;
   1:  PR[91,3] = PR[90,3] + 84.871;
   1:L PR[91] R[100]mm/sec CNT100;
   1:  PR[91,1] = PR[90,1] + -50.363;
   1:  PR[91,2] = PR[90,2] + -19.646;
   1:  PR[91,3] = PR[90,3] + 84.881;
   1:L PR[91] R[100]mm/sec CNT100;
   1:  PR[91,1] = PR[90,1] + -45.579;
   1:  PR[91,2] = PR[90,2] + -22.133;
   1:  PR[91,3] = PR[90,3] + 84.892;
   1:L PR[91] R[100]mm/sec CNT100;
   1:  PR[91,1] = PR[90,1] + -39.579;
   1:  PR[91,2] = PR[90,2] + -23.958;
   1:  PR[91,3] = PR[90,3] + 84.915;
   1:L PR[91] R[100]mm/sec CNT100;
   1:  PR[91,1] = PR[90,1] + -36.288;
   1:  PR[91,2] = PR[90,2] + -24.911;
   1:  PR[91,3] = PR[90,3] + 84.941;
   1:L PR[91] R[100]mm/sec CNT100;
   1:  PR[91,1] = PR[90,1] + -33.240;
   1:  PR[91,2] = PR[90,2] + -25.503;
   1:  PR[91,3] = PR[90,3] + 84.955;
   1:L PR[91] R[100]mm/sec CNT100;
   1:  PR[91,1] = PR[90,1] + -27.855;
   1:  PR[91,2] = PR[90,2] + -26.462;
   1:  PR[91,3] = PR[90,3] + 84.968;
   1:L PR[91] R[100]mm/sec CNT100;
   1:  PR[91,1] = PR[90,1] + -18.268;
   1:  PR[91,2] = PR[90,2] + -27.470;
   1:  PR[91,3] = PR[90,3] + 84.991;
   1:L PR[91] R[100]mm/sec CNT100;
   1:  PR[91,1] = PR[90,1] + -13.610;
   1:  PR[91,2] = PR[90,2] + -27.649;
   1:  PR[91,3] = PR[90,3] + 85.031;
   1:L PR[91] R[100]mm/sec CNT100;
   1:  PR[91,1] = PR[90,1] + -8.222;
   1:  PR[91,2] = PR[90,2] + -27.828;
   1:  PR[91,3] = PR[90,3] + 85.051;
   1:L PR[91] R[100]mm/sec CNT100;
   1:  PR[91,1] = PR[90,1] + -0.378;
   1:  PR[91,2] = PR[90,2] + -27.581;
   1:  PR[91,3] = PR[90,3] + 85.073;
   1:L PR[91] R[100]mm/sec CNT100;
   1:  PR[91,1] = PR[90,1] + 2.123;
   1:  PR[91,2] = PR[90,2] + -27.487;
   1:  PR[91,3] = PR[90,3] + 85.106;
   1:L PR[91] R[100]mm/sec CNT100;
   1:  PR[91,1] = PR[90,1] + 2.862;
   1:  PR[91,2] = PR[90,2] + -27.436;
   1:  PR[91,3] = PR[90,3] + 85.116;
   1:L PR[91] R[100]mm/sec CNT100;
   1:  PR[91,1] = PR[90,1] + 3.357;
   1:  PR[91,2] = PR[90,2] + -27.468;
   1:  PR[91,3] = PR[90,3] + 85.119;
   1:L PR[91] R[100]mm/sec CNT100;
   1:  PR[91,1] = PR[90,1] + 7.999;
   1:  PR[91,2] = PR[90,2] + -27.526;
   1:  PR[91,3] = PR[90,3] + 85.122;
   1:L PR[91] R[100]mm/sec CNT100;
   1:  PR[91,1] = PR[90,1] + 8.784;
   1:  PR[91,2] = PR[90,2] + -27.509;
   1:  PR[91,3] = PR[90,3] + 85.141;
   1:L PR[91] R[100]mm/sec CNT100;
   1:  PR[91,1] = PR[90,1] + 10.312;
   1:  PR[91,2] = PR[90,2] + -27.406;
   1:  PR[91,3] = PR[90,3] + 85.144;
   1:L PR[91] R[100]mm/sec CNT100;
   1:  PR[91,1] = PR[90,1] + 12.488;
   1:  PR[91,2] = PR[90,2] + -27.206;
   1:  PR[91,3] = PR[90,3] + 85.151;
   1:L PR[91] R[100]mm/sec CNT100;
   1:  PR[91,1] = PR[90,1] + 14.691;
   1:  PR[91,2] = PR[90,2] + -27.574;
   1:  PR[91,3] = PR[90,3] + 85.160;
   1:L PR[91] R[100]mm/sec CNT100;
   1:  PR[91,1] = PR[90,1] + 17.503;
   1:  PR[91,2] = PR[90,2] + -27.919;
   1:  PR[91,3] = PR[90,3] + 85.169;
   1:L PR[91] R[100]mm/sec CNT100;
   1:  PR[91,1] = PR[90,1] + 19.520;
   1:  PR[91,2] = PR[90,2] + -27.850;
   1:  PR[91,3] = PR[90,3] + 85.181;
   1:L PR[91] R[100]mm/sec CNT100;
   1:  PR[91,1] = PR[90,1] + 22.617;
   1:  PR[91,2] = PR[90,2] + -27.793;
   1:  PR[91,3] = PR[90,3] + 85.189;
   1:L PR[91] R[100]mm/sec CNT100;
   1:  PR[91,1] = PR[90,1] + 25.077;
   1:  PR[91,2] = PR[90,2] + -28.382;
   1:  PR[91,3] = PR[90,3] + 85.202;
   1:L PR[91] R[100]mm/sec CNT100;
   1:  PR[91,1] = PR[90,1] + 26.255;
   1:  PR[91,2] = PR[90,2] + -28.638;
   1:  PR[91,3] = PR[90,3] + 85.213;
   1:L PR[91] R[100]mm/sec CNT100;
   1:  PR[91,1] = PR[90,1] + 28.183;
   1:  PR[91,2] = PR[90,2] + -29.086;
   1:  PR[91,3] = PR[90,3] + 85.218;
   1:L PR[91] R[100]mm/sec CNT100;
   1:  PR[91,1] = PR[90,1] + 33.328;
   1:  PR[91,2] = PR[90,2] + -29.386;
   1:  PR[91,3] = PR[90,3] + 85.226;
   1:L PR[91] R[100]mm/sec CNT100;
   1:  PR[91,1] = PR[90,1] + 35.825;
   1:  PR[91,2] = PR[90,2] + -29.084;
   1:  PR[91,3] = PR[90,3] + 85.247;
   1:L PR[91] R[100]mm/sec CNT100;
   1:  PR[91,1] = PR[90,1] + 38.494;
   1:  PR[91,2] = PR[90,2] + -28.783;
   1:  PR[91,3] = PR[90,3] + 85.258;
   1:L PR[91] R[100]mm/sec CNT100;
   1:  PR[91,1] = PR[90,1] + 39.496;
   1:  PR[91,2] = PR[90,2] + -28.506;
   1:  PR[91,3] = PR[90,3] + 85.269;
   1:L PR[91] R[100]mm/sec CNT100;
   1:  PR[91,1] = PR[90,1] + 43.463;
   1:  PR[91,2] = PR[90,2] + -27.362;
   1:  PR[91,3] = PR[90,3] + 85.273;
   1:L PR[91] R[100]mm/sec CNT100;
   1:  PR[91,1] = PR[90,1] + 48.032;
   1:  PR[91,2] = PR[90,2] + -25.178;
   1:  PR[91,3] = PR[90,3] + 85.291;
   1:L PR[91] R[100]mm/sec CNT100;
   1:  PR[91,1] = PR[90,1] + 49.734;
   1:  PR[91,2] = PR[90,2] + -23.962;
   1:  PR[91,3] = PR[90,3] + 85.312;
   1:L PR[91] R[100]mm/sec CNT100;
   1:  PR[91,1] = PR[90,1] + 51.975;
   1:  PR[91,2] = PR[90,2] + -22.551;
   1:  PR[91,3] = PR[90,3] + 85.321;
   1:L PR[91] R[100]mm/sec CNT100;
   1:  PR[91,1] = PR[90,1] + 52.913;
   1:  PR[91,2] = PR[90,2] + -21.851;
   1:  PR[91,3] = PR[90,3] + 85.332;
   1:L PR[91] R[100]mm/sec CNT100;
   1:  PR[91,1] = PR[90,1] + 54.901;
   1:  PR[91,2] = PR[90,2] + -20.057;
   1:  PR[91,3] = PR[90,3] + 85.336;
   1:L PR[91] R[100]mm/sec CNT100;
   1:  PR[91,1] = PR[90,1] + 57.147;
   1:  PR[91,2] = PR[90,2] + -17.716;
   1:  PR[91,3] = PR[90,3] + 85.348;
   1:L PR[91] R[100]mm/sec CNT100;
   1:  PR[91,1] = PR[90,1] + 57.233;
   1:  PR[91,2] = PR[90,2] + -17.604;
   1:  PR[91,3] = PR[90,3] + 85.361;
   1:L PR[91] R[100]mm/sec CNT100;
   1:  PR[91,1] = PR[90,1] + 57.549;
   1:  PR[91,2] = PR[90,2] + -17.139;
   1:  PR[91,3] = PR[90,3] + 85.362;
   1:L PR[91] R[100]mm/sec CNT100;
   1:  PR[91,1] = PR[90,1] + 59.784;
   1:  PR[91,2] = PR[90,2] + -14.469;
   1:  PR[91,3] = PR[90,3] + 85.364;
   1:L PR[91] R[100]mm/sec CNT100;
   1:  PR[91,1] = PR[90,1] + 60.799;
   1:  PR[91,2] = PR[90,2] + -13.045;
   1:  PR[91,3] = PR[90,3] + 85.379;
   1:L PR[91] R[100]mm/sec CNT100;
   1:  PR[91,1] = PR[90,1] + 61.561;
   1:  PR[91,2] = PR[90,2] + -11.686;
   1:  PR[91,3] = PR[90,3] + 85.386;
   1:L PR[91] R[100]mm/sec CNT100;
   1:  PR[91,1] = PR[90,1] + 62.905;
   1:  PR[91,2] = PR[90,2] + -8.916;
   1:  PR[91,3] = PR[90,3] + 85.392;
   1:L PR[91] R[100]mm/sec CNT100;
   1:  PR[91,1] = PR[90,1] + 63.054;
   1:  PR[91,2] = PR[90,2] + -8.651;
   1:  PR[91,3] = PR[90,3] + 85.405;
   1:L PR[91] R[100]mm/sec CNT100;
   1:  PR[91,1] = PR[90,1] + 64.327;
   1:  PR[91,2] = PR[90,2] + -4.746;
   1:  PR[91,3] = PR[90,3] + 85.407;
   1:L PR[91] R[100]mm/sec CNT100;
   1:  PR[91,1] = PR[90,1] + 64.762;
   1:  PR[91,2] = PR[90,2] + -0.729;
   1:  PR[91,3] = PR[90,3] + 85.424;
   1:L PR[91] R[100]mm/sec CNT100;
   1:  PR[91,1] = PR[90,1] + 64.327;
   1:  PR[91,2] = PR[90,2] + 3.287;
   1:  PR[91,3] = PR[90,3] + 85.441;
   1:L PR[91] R[100]mm/sec CNT100;
   1:  PR[91,1] = PR[90,1] + 63.054;
   1:  PR[91,2] = PR[90,2] + 7.192;
   1:  PR[91,3] = PR[90,3] + 85.457;
   1:L PR[91] R[100]mm/sec CNT100;
   1:  PR[91,1] = PR[90,1] + 62.905;
   1:  PR[91,2] = PR[90,2] + 7.457;
   1:  PR[91,3] = PR[90,3] + 85.474;
   1:L PR[91] R[100]mm/sec CNT100;
   1:  PR[91,1] = PR[90,1] + 61.561;
   1:  PR[91,2] = PR[90,2] + 10.227;
   1:  PR[91,3] = PR[90,3] + 85.476;
   1:L PR[91] R[100]mm/sec CNT100;
   1:  PR[91,1] = PR[90,1] + 60.799;
   1:  PR[91,2] = PR[90,2] + 11.587;
   1:  PR[91,3] = PR[90,3] + 85.489;
   1:L PR[91] R[100]mm/sec CNT100;
   1:  PR[91,1] = PR[90,1] + 59.784;
   1:  PR[91,2] = PR[90,2] + 13.010;
   1:  PR[91,3] = PR[90,3] + 85.495;
   1:L PR[91] R[100]mm/sec CNT100;
   1:  PR[91,1] = PR[90,1] + 57.549;
   1:  PR[91,2] = PR[90,2] + 15.680;
   1:  PR[91,3] = PR[90,3] + 85.502;
   1:L PR[91] R[100]mm/sec CNT100;
   1:  PR[91,1] = PR[90,1] + 57.233;
   1:  PR[91,2] = PR[90,2] + 16.145;
   1:  PR[91,3] = PR[90,3] + 85.517;
   1:L PR[91] R[100]mm/sec CNT100;
   1:  PR[91,1] = PR[90,1] + 57.147;
   1:  PR[91,2] = PR[90,2] + 16.257;
   1:  PR[91,3] = PR[90,3] + 85.519;
   1:L PR[91] R[100]mm/sec CNT100;
   1:  PR[91,1] = PR[90,1] + 54.901;
   1:  PR[91,2] = PR[90,2] + 18.599;
   1:  PR[91,3] = PR[90,3] + 85.520;
   1:L PR[91] R[100]mm/sec CNT100;
   1:  PR[91,1] = PR[90,1] + 52.913;
   1:  PR[91,2] = PR[90,2] + 20.392;
   1:  PR[91,3] = PR[90,3] + 85.533;
   1:L PR[91] R[100]mm/sec CNT100;
   1:  PR[91,1] = PR[90,1] + 51.975;
   1:  PR[91,2] = PR[90,2] + 21.092;
   1:  PR[91,3] = PR[90,3] + 85.545;
   1:L PR[91] R[100]mm/sec CNT100;
   1:  PR[91,1] = PR[90,1] + 49.734;
   1:  PR[91,2] = PR[90,2] + 22.503;
   1:  PR[91,3] = PR[90,3] + 85.549;
   1:L PR[91] R[100]mm/sec CNT100;
   1:  PR[91,1] = PR[90,1] + 48.032;
   1:  PR[91,2] = PR[90,2] + 23.719;
   1:  PR[91,3] = PR[90,3] + 85.560;
   1:L PR[91] R[100]mm/sec CNT100;
   1:  PR[91,1] = PR[90,1] + 43.463;
   1:  PR[91,2] = PR[90,2] + 25.903;
   1:  PR[91,3] = PR[90,3] + 85.569;
   1:L PR[91] R[100]mm/sec CNT100;
   1:  PR[91,1] = PR[90,1] + 39.496;
   1:  PR[91,2] = PR[90,2] + 27.047;
   1:  PR[91,3] = PR[90,3] + 85.590;
   1:L PR[91] R[100]mm/sec CNT100;
   1:  PR[91,1] = PR[90,1] + 38.494;
   1:  PR[91,2] = PR[90,2] + 27.324;
   1:  PR[91,3] = PR[90,3] + 85.608;
   1:L PR[91] R[100]mm/sec CNT100;
   1:  PR[91,1] = PR[90,1] + 35.825;
   1:  PR[91,2] = PR[90,2] + 27.625;
   1:  PR[91,3] = PR[90,3] + 85.612;
   1:L PR[91] R[100]mm/sec CNT100;
   1:  PR[91,1] = PR[90,1] + 33.328;
   1:  PR[91,2] = PR[90,2] + 27.927;
   1:  PR[91,3] = PR[90,3] + 85.623;
   1:L PR[91] R[100]mm/sec CNT100;
   1:  PR[91,1] = PR[90,1] + 28.183;
   1:  PR[91,2] = PR[90,2] + 27.627;
   1:  PR[91,3] = PR[90,3] + 85.634;
   1:L PR[91] R[100]mm/sec CNT100;
   1:  PR[91,1] = PR[90,1] + 26.255;
   1:  PR[91,2] = PR[90,2] + 27.179;
   1:  PR[91,3] = PR[90,3] + 85.655;
   1:L PR[91] R[100]mm/sec CNT100;
   1:  PR[91,1] = PR[90,1] + 25.077;
   1:  PR[91,2] = PR[90,2] + 26.923;
   1:  PR[91,3] = PR[90,3] + 85.663;
   1:L PR[91] R[100]mm/sec CNT100;
   1:  PR[91,1] = PR[90,1] + 22.600;
   1:  PR[91,2] = PR[90,2] + 26.330;
   1:  PR[91,3] = PR[90,3] + 85.668;
   1:L PR[91] R[100]mm/sec CNT100;
   1:  PR[91,1] = PR[90,1] + 20.421;
   1:  PR[91,2] = PR[90,2] + 26.408;
   1:  PR[91,3] = PR[90,3] + 85.679;
   1:L PR[91] R[100]mm/sec CNT100;
   1:  PR[91,1] = PR[90,1] + 17.519;
   1:  PR[91,2] = PR[90,2] + 26.462;
   1:  PR[91,3] = PR[90,3] + 85.688;
   1:L PR[91] R[100]mm/sec CNT100;
   1:  PR[91,1] = PR[90,1] + 14.694;
   1:  PR[91,2] = PR[90,2] + 26.116;
   1:  PR[91,3] = PR[90,3] + 85.700;
   1:L PR[91] R[100]mm/sec CNT100;
   1:  PR[91,1] = PR[90,1] + 12.488;
   1:  PR[91,2] = PR[90,2] + 25.747;
   1:  PR[91,3] = PR[90,3] + 85.712;
   1:L PR[91] R[100]mm/sec CNT100;
   1:  PR[91,1] = PR[90,1] + 10.311;
   1:  PR[91,2] = PR[90,2] + 25.948;
   1:  PR[91,3] = PR[90,3] + 85.721;
   1:L PR[91] R[100]mm/sec CNT100;
   1:  PR[91,1] = PR[90,1] + 8.810;
   1:  PR[91,2] = PR[90,2] + 26.049;
   1:  PR[91,3] = PR[90,3] + 85.731;
   1:L PR[91] R[100]mm/sec CNT100;
   1:  PR[91,1] = PR[90,1] + 3.401;
   1:  PR[91,2] = PR[90,2] + 26.009;
   1:  PR[91,3] = PR[90,3] + 85.737;
   1:L PR[91] R[100]mm/sec CNT100;
   1:  PR[91,1] = PR[90,1] + 2.940;
   1:  PR[91,2] = PR[90,2] + 25.963;
   1:  PR[91,3] = PR[90,3] + 85.759;
   1:L PR[91] R[100]mm/sec CNT100;
   1:  PR[91,1] = PR[90,1] + 2.522;
   1:  PR[91,2] = PR[90,2] + 26.001;
   1:  PR[91,3] = PR[90,3] + 85.761;
   1:L PR[91] R[100]mm/sec CNT100;
   1:  PR[91,1] = PR[90,1] + -0.383;
   1:  PR[91,2] = PR[90,2] + 26.122;
   1:  PR[91,3] = PR[90,3] + 85.763;
   1:L PR[91] R[100]mm/sec CNT100;
   1:  PR[91,1] = PR[90,1] + -8.222;
   1:  PR[91,2] = PR[90,2] + 26.369;
   1:  PR[91,3] = PR[90,3] + 85.775;
   1:L PR[91] R[100]mm/sec CNT100;
   1:  PR[91,1] = PR[90,1] + -13.610;
   1:  PR[91,2] = PR[90,2] + 26.190;
   1:  PR[91,3] = PR[90,3] + 85.808;
   1:L PR[91] R[100]mm/sec CNT100;
   1:  PR[91,1] = PR[90,1] + -18.268;
   1:  PR[91,2] = PR[90,2] + 26.011;
   1:  PR[91,3] = PR[90,3] + 85.830;
   1:L PR[91] R[100]mm/sec CNT100;
   1:  PR[91,1] = PR[90,1] + -27.855;
   1:  PR[91,2] = PR[90,2] + 25.003;
   1:  PR[91,3] = PR[90,3] + 85.850;
   1:L PR[91] R[100]mm/sec CNT100;
   1:  PR[91,1] = PR[90,1] + -33.241;
   1:  PR[91,2] = PR[90,2] + 24.044;
   1:  PR[91,3] = PR[90,3] + 85.890;
   1:L PR[91] R[100]mm/sec CNT100;
   1:  PR[91,1] = PR[90,1] + -36.397;
   1:  PR[91,2] = PR[90,2] + 23.433;
   1:  PR[91,3] = PR[90,3] + 85.913;
   1:L PR[91] R[100]mm/sec CNT100;
   1:  PR[91,1] = PR[90,1] + -44.365;
   1:  PR[91,2] = PR[90,2] + 21.053;
   1:  PR[91,3] = PR[90,3] + 85.926;
   1:L PR[91] R[100]mm/sec CNT100;
   1:  PR[91,1] = PR[90,1] + -45.496;
   1:  PR[91,2] = PR[90,2] + 20.675;
   1:  PR[91,3] = PR[90,3] + 85.961;
   1:L PR[91] R[100]mm/sec CNT100;
   1:  PR[91,1] = PR[90,1] + -46.798;
   1:  PR[91,2] = PR[90,2] + 20.047;
   1:  PR[91,3] = PR[90,3] + 85.966;
   1:L PR[91] R[100]mm/sec CNT100;
   1:  PR[91,1] = PR[90,1] + -51.729;
   1:  PR[91,2] = PR[90,2] + 17.534;
   1:  PR[91,3] = PR[90,3] + 85.972;
   1:L PR[91] R[100]mm/sec CNT100;
   1:  PR[91] = PR[90];
   1:  PR[91,1] = PR[90,1] + -54.557;
   1:  PR[91,2] = PR[90,2] + 14.545;
   1:  PR[91,3] = PR[90,3] + 87.295;
   1:L PR[91] R[100]mm/sec CNT100;
   1:  PR[91,1] = PR[90,1] + -55.732;
   1:  PR[91,2] = PR[90,2] + 13.660;
   1:  PR[91,3] = PR[90,3] + 86.017;
   1:L PR[91] R[100]mm/sec CNT100;
   1:  PR[91,1] = PR[90,1] + -57.619;
   1:  PR[91,2] = PR[90,2] + 11.580;
   1:  PR[91,3] = PR[90,3] + 86.023;
   1:L PR[91] R[100]mm/sec CNT100;
   1:  PR[91,1] = PR[90,1] + -59.303;
   1:  PR[91,2] = PR[90,2] + 9.513;
   1:  PR[91,3] = PR[90,3] + 86.035;
   1:L PR[91] R[100]mm/sec CNT100;
   1:  PR[91,1] = PR[90,1] + -59.600;
   1:  PR[91,2] = PR[90,2] + 9.136;
   1:  PR[91,3] = PR[90,3] + 86.046;
   1:L PR[91] R[100]mm/sec CNT100;
   1:  PR[91,1] = PR[90,1] + -61.331;
   1:  PR[91,2] = PR[90,2] + 5.370;
   1:  PR[91,3] = PR[90,3] + 86.048;
   1:L PR[91] R[100]mm/sec CNT100;
   1:  PR[91,1] = PR[90,1] + -61.838;
   1:  PR[91,2] = PR[90,2] + 4.232;
   1:  PR[91,3] = PR[90,3] + 86.066;
   1:L PR[91] R[100]mm/sec CNT100;
   1:  PR[91,1] = PR[90,1] + -62.067;
   1:  PR[91,2] = PR[90,2] + 2.669;
   1:  PR[91,3] = PR[90,3] + 86.071;
   1:L PR[91] R[100]mm/sec CNT100;
   1:  PR[91,1] = PR[90,1] + -62.370;
   1:  PR[91,2] = PR[90,2] + 1.388;
   1:  PR[91,3] = PR[90,3] + 86.077;
   1:L PR[91] R[100]mm/sec CNT100;
   1:  PR[91,1] = PR[90,1] + -62.716;
   1:  PR[91,2] = PR[90,2] + -0.626;
   1:  PR[91,3] = PR[90,3] + 86.083;
   1:L PR[91] R[100]mm/sec CNT100;
   1:  PR[91,1] = PR[90,1] + -62.606;
   1:  PR[91,2] = PR[90,2] + -1.023;
   1:  PR[91,3] = PR[90,3] + 86.092;
   1:L PR[91] R[100]mm/sec CNT100;
   1:  PR[91,1] = PR[90,1] + -62.021;
   1:  PR[91,2] = PR[90,2] + -5.413;
   1:  PR[91,3] = PR[90,3] + 86.093;
   1:L PR[91] R[100]mm/sec CNT100;
   1:  PR[91,1] = PR[90,1] + -60.584;
   1:  PR[91,2] = PR[90,2] + -8.897;
   1:  PR[91,3] = PR[90,3] + 86.112;
   1:L PR[91] R[100]mm/sec CNT100;
   1:  PR[91,1] = PR[90,1] + -60.130;
   1:  PR[91,2] = PR[90,2] + -9.863;
   1:  PR[91,3] = PR[90,3] + 86.128;
   1:L PR[91] R[100]mm/sec CNT100;
   1:  PR[91,1] = PR[90,1] + -57.250;
   1:  PR[91,2] = PR[90,2] + -13.376;
   1:  PR[91,3] = PR[90,3] + 86.132;
   1:L PR[91] R[100]mm/sec CNT100;
   1:  PR[91,1] = PR[90,1] + -56.430;
   1:  PR[91,2] = PR[90,2] + -14.341;
   1:  PR[91,3] = PR[90,3] + 86.152;
   1:L PR[91] R[100]mm/sec CNT100;
   1:  PR[91,1] = PR[90,1] + -53.694;
   1:  PR[91,2] = PR[90,2] + -16.543;
   1:  PR[91,3] = PR[90,3] + 86.157;
   1:L PR[91] R[100]mm/sec CNT100;
   1:  PR[91,1] = PR[90,1] + -51.020;
   1:  PR[91,2] = PR[90,2] + -18.600;
   1:  PR[91,3] = PR[90,3] + 86.172;
   1:L PR[91] R[100]mm/sec CNT100;
   1:  PR[91,1] = PR[90,1] + -49.545;
   1:  PR[91,2] = PR[90,2] + -19.415;
   1:  PR[91,3] = PR[90,3] + 86.186;
   1:L PR[91] R[100]mm/sec CNT100;
   1:  PR[91,1] = PR[90,1] + -46.306;
   1:  PR[91,2] = PR[90,2] + -21.100;
   1:  PR[91,3] = PR[90,3] + 86.193;
   1:L PR[91] R[100]mm/sec CNT100;
   1:  PR[91,1] = PR[90,1] + -44.275;
   1:  PR[91,2] = PR[90,2] + -22.033;
   1:  PR[91,3] = PR[90,3] + 86.209;
   1:L PR[91] R[100]mm/sec CNT100;
   1:  PR[91,1] = PR[90,1] + -43.151;
   1:  PR[91,2] = PR[90,2] + -22.468;
   1:  PR[91,3] = PR[90,3] + 86.218;
   1:L PR[91] R[100]mm/sec CNT100;
   1:  PR[91,1] = PR[90,1] + -38.587;
   1:  PR[91,2] = PR[90,2] + -23.856;
   1:  PR[91,3] = PR[90,3] + 86.223;
   1:L PR[91] R[100]mm/sec CNT100;
   1:  PR[91,1] = PR[90,1] + -34.294;
   1:  PR[91,2] = PR[90,2] + -25.099;
   1:  PR[91,3] = PR[90,3] + 86.243;
   1:L PR[91] R[100]mm/sec CNT100;
   1:  PR[91,1] = PR[90,1] + -25.383;
   1:  PR[91,2] = PR[90,2] + -26.694;
   1:  PR[91,3] = PR[90,3] + 86.262;
   1:L PR[91] R[100]mm/sec CNT100;
   1:  PR[91,1] = PR[90,1] + -15.722;
   1:  PR[91,2] = PR[90,2] + -27.714;
   1:  PR[91,3] = PR[90,3] + 86.300;
   1:L PR[91] R[100]mm/sec CNT100;
   1:  PR[91,1] = PR[90,1] + -10.070;
   1:  PR[91,2] = PR[90,2] + -27.932;
   1:  PR[91,3] = PR[90,3] + 86.341;
   1:L PR[91] R[100]mm/sec CNT100;
   1:  PR[91,1] = PR[90,1] + -5.595;
   1:  PR[91,2] = PR[90,2] + -28.081;
   1:  PR[91,3] = PR[90,3] + 86.365;
   1:L PR[91] R[100]mm/sec CNT100;
   1:  PR[91,1] = PR[90,1] + 3.264;
   1:  PR[91,2] = PR[90,2] + -27.801;
   1:  PR[91,3] = PR[90,3] + 86.384;
   1:L PR[91] R[100]mm/sec CNT100;
   1:  PR[91,1] = PR[90,1] + 5.227;
   1:  PR[91,2] = PR[90,2] + -27.718;
   1:  PR[91,3] = PR[90,3] + 86.422;
   1:L PR[91] R[100]mm/sec CNT100;
   1:  PR[91,1] = PR[90,1] + 8.583;
   1:  PR[91,2] = PR[90,2] + -27.766;
   1:  PR[91,3] = PR[90,3] + 86.430;
   1:L PR[91] R[100]mm/sec CNT100;
   1:  PR[91,1] = PR[90,1] + 9.829;
   1:  PR[91,2] = PR[90,2] + -27.740;
   1:  PR[91,3] = PR[90,3] + 86.444;
   1:L PR[91] R[100]mm/sec CNT100;
   1:  PR[91,1] = PR[90,1] + 11.028;
   1:  PR[91,2] = PR[90,2] + -27.673;
   1:  PR[91,3] = PR[90,3] + 86.449;
   1:L PR[91] R[100]mm/sec CNT100;
   1:  PR[91,1] = PR[90,1] + 13.197;
   1:  PR[91,2] = PR[90,2] + -27.489;
   1:  PR[91,3] = PR[90,3] + 86.454;
   1:L PR[91] R[100]mm/sec CNT100;
   1:  PR[91,1] = PR[90,1] + 14.197;
   1:  PR[91,2] = PR[90,2] + -27.656;
   1:  PR[91,3] = PR[90,3] + 86.464;
   1:L PR[91] R[100]mm/sec CNT100;
   1:  PR[91,1] = PR[90,1] + 17.715;
   1:  PR[91,2] = PR[90,2] + -28.088;
   1:  PR[91,3] = PR[90,3] + 86.468;
   1:L PR[91] R[100]mm/sec CNT100;
   1:  PR[91,1] = PR[90,1] + 18.395;
   1:  PR[91,2] = PR[90,2] + -28.064;
   1:  PR[91,3] = PR[90,3] + 86.483;
   1:L PR[91] R[100]mm/sec CNT100;
   1:  PR[91,1] = PR[90,1] + 22.306;
   1:  PR[91,2] = PR[90,2] + -27.992;
   1:  PR[91,3] = PR[90,3] + 86.486;
   1:L PR[91] R[100]mm/sec CNT100;
   1:  PR[91,1] = PR[90,1] + 23.329;
   1:  PR[91,2] = PR[90,2] + -28.237;
   1:  PR[91,3] = PR[90,3] + 86.502;
   1:L PR[91] R[100]mm/sec CNT100;
   1:  PR[91,1] = PR[90,1] + 25.049;
   1:  PR[91,2] = PR[90,2] + -28.611;
   1:  PR[91,3] = PR[90,3] + 86.507;
   1:L PR[91] R[100]mm/sec CNT100;
   1:  PR[91,1] = PR[90,1] + 27.930;
   1:  PR[91,2] = PR[90,2] + -29.280;
   1:  PR[91,3] = PR[90,3] + 86.514;
   1:L PR[91] R[100]mm/sec CNT100;
   1:  PR[91,1] = PR[90,1] + 33.107;
   1:  PR[91,2] = PR[90,2] + -29.577;
   1:  PR[91,3] = PR[90,3] + 86.527;
   1:L PR[91] R[100]mm/sec CNT100;
   1:  PR[91,1] = PR[90,1] + 38.187;
   1:  PR[91,2] = PR[90,2] + -28.964;
   1:  PR[91,3] = PR[90,3] + 86.548;
   1:L PR[91] R[100]mm/sec CNT100;
   1:  PR[91,1] = PR[90,1] + 38.984;
   1:  PR[91,2] = PR[90,2] + -28.719;
   1:  PR[91,3] = PR[90,3] + 86.570;
   1:L PR[91] R[100]mm/sec CNT100;
   1:  PR[91,1] = PR[90,1] + 43.191;
   1:  PR[91,2] = PR[90,2] + -27.507;
   1:  PR[91,3] = PR[90,3] + 86.574;
   1:L PR[91] R[100]mm/sec CNT100;
   1:  PR[91,1] = PR[90,1] + 47.791;
   1:  PR[91,2] = PR[90,2] + -25.296;
   1:  PR[91,3] = PR[90,3] + 86.592;
   1:L PR[91] R[100]mm/sec CNT100;
   1:  PR[91,1] = PR[90,1] + 51.906;
   1:  PR[91,2] = PR[90,2] + -22.353;
   1:  PR[91,3] = PR[90,3] + 86.614;
   1:L PR[91] R[100]mm/sec CNT100;
   1:  PR[91,1] = PR[90,1] + 55.009;
   1:  PR[91,2] = PR[90,2] + -19.554;
   1:  PR[91,3] = PR[90,3] + 86.635;
   1:L PR[91] R[100]mm/sec CNT100;
   1:  PR[91,1] = PR[90,1] + 56.295;
   1:  PR[91,2] = PR[90,2] + -18.214;
   1:  PR[91,3] = PR[90,3] + 86.653;
   1:L PR[91] R[100]mm/sec CNT100;
   1:  PR[91,1] = PR[90,1] + 57.361;
   1:  PR[91,2] = PR[90,2] + -16.831;
   1:  PR[91,3] = PR[90,3] + 86.660;
   1:L PR[91] R[100]mm/sec CNT100;
   1:  PR[91,1] = PR[90,1] + 59.192;
   1:  PR[91,2] = PR[90,2] + -14.135;
   1:  PR[91,3] = PR[90,3] + 86.668;
   1:L PR[91] R[100]mm/sec CNT100;
   1:  PR[91,1] = PR[90,1] + 59.505;
   1:  PR[91,2] = PR[90,2] + -13.760;
   1:  PR[91,3] = PR[90,3] + 86.682;
   1:L PR[91] R[100]mm/sec CNT100;
   1:  PR[91,1] = PR[90,1] + 59.548;
   1:  PR[91,2] = PR[90,2] + -13.700;
   1:  PR[91,3] = PR[90,3] + 86.684;
   1:L PR[91] R[100]mm/sec CNT100;
   1:  PR[91,1] = PR[90,1] + 61.254;
   1:  PR[91,2] = PR[90,2] + -10.656;
   1:L PR[91] R[100]mm/sec CNT100;
   1:  PR[91,1] = PR[90,1] + 61.997;
   1:  PR[91,2] = PR[90,2] + -9.125;
   1:  PR[91,3] = PR[90,3] + 86.699;
   1:L PR[91] R[100]mm/sec CNT100;
   1:  PR[91,1] = PR[90,1] + 62.495;
   1:  PR[91,2] = PR[90,2] + -7.575;
   1:  PR[91,3] = PR[90,3] + 86.706;
   1:L PR[91] R[100]mm/sec CNT100;
   1:  PR[91,1] = PR[90,1] + 63.268;
   1:  PR[91,2] = PR[90,2] + -4.845;
   1:  PR[91,3] = PR[90,3] + 86.713;
   1:L PR[91] R[100]mm/sec CNT100;
   1:  PR[91,1] = PR[90,1] + 63.661;
   1:  PR[91,2] = PR[90,2] + -0.729;
   1:  PR[91,3] = PR[90,3] + 86.725;
   1:L PR[91] R[100]mm/sec CNT100;
   1:  PR[91,1] = PR[90,1] + 63.268;
   1:  PR[91,2] = PR[90,2] + 3.386;
   1:  PR[91,3] = PR[90,3] + 86.742;
   1:L PR[91] R[100]mm/sec CNT100;
   1:  PR[91,1] = PR[90,1] + 62.495;
   1:  PR[91,2] = PR[90,2] + 6.116;
   1:  PR[91,3] = PR[90,3] + 86.760;
   1:L PR[91] R[100]mm/sec CNT100;
   1:  PR[91,1] = PR[90,1] + 61.997;
   1:  PR[91,2] = PR[90,2] + 7.666;
   1:  PR[91,3] = PR[90,3] + 86.772;
   1:L PR[91] R[100]mm/sec CNT100;
   1:  PR[91,1] = PR[90,1] + 61.254;
   1:  PR[91,2] = PR[90,2] + 9.197;
   1:  PR[91,3] = PR[90,3] + 86.778;
   1:L PR[91] R[100]mm/sec CNT100;
   1:  PR[91,1] = PR[90,1] + 59.548;
   1:  PR[91,2] = PR[90,2] + 12.241;
   1:  PR[91,3] = PR[90,3] + 86.786;
   1:L PR[91] R[100]mm/sec CNT100;
   1:  PR[91,1] = PR[90,1] + 59.505;
   1:  PR[91,2] = PR[90,2] + 12.302;
   1:  PR[91,3] = PR[90,3] + 86.800;
   1:L PR[91] R[100]mm/sec CNT100;
   1:  PR[91,1] = PR[90,1] + 59.192;
   1:  PR[91,2] = PR[90,2] + 12.676;
   1:  PR[91,3] = PR[90,3] + 86.801;
   1:L PR[91] R[100]mm/sec CNT100;
   1:  PR[91,1] = PR[90,1] + 57.361;
   1:  PR[91,2] = PR[90,2] + 15.372;
   1:  PR[91,3] = PR[90,3] + 86.803;
   1:L PR[91] R[100]mm/sec CNT100;
   1:  PR[91,1] = PR[90,1] + 56.295;
   1:  PR[91,2] = PR[90,2] + 16.755;
   1:  PR[91,3] = PR[90,3] + 86.816;
   1:L PR[91] R[100]mm/sec CNT100;
   1:  PR[91,1] = PR[90,1] + 55.009;
   1:  PR[91,2] = PR[90,2] + 18.095;
   1:  PR[91,3] = PR[90,3] + 86.824;
   1:L PR[91] R[100]mm/sec CNT100;
   1:  PR[91,1] = PR[90,1] + 51.901;
   1:  PR[91,2] = PR[90,2] + 20.899;
   1:  PR[91,3] = PR[90,3] + 86.832;
   1:L PR[91] R[100]mm/sec CNT100;
   1:  PR[91,1] = PR[90,1] + 47.791;
   1:  PR[91,2] = PR[90,2] + 23.837;
   1:  PR[91,3] = PR[90,3] + 86.849;
   1:L PR[91] R[100]mm/sec CNT100;
   1:  PR[91,1] = PR[90,1] + 43.191;
   1:  PR[91,2] = PR[90,2] + 26.048;
   1:  PR[91,3] = PR[90,3] + 86.871;
   1:L PR[91] R[100]mm/sec CNT100;
   1:  PR[91,1] = PR[90,1] + 38.984;
   1:  PR[91,2] = PR[90,2] + 27.261;
   1:  PR[91,3] = PR[90,3] + 86.892;
   1:L PR[91] R[100]mm/sec CNT100;
   1:  PR[91,1] = PR[90,1] + 38.187;
   1:  PR[91,2] = PR[90,2] + 27.505;
   1:  PR[91,3] = PR[90,3] + 86.911;
   1:L PR[91] R[100]mm/sec CNT100;
   1:  PR[91,1] = PR[90,1] + 33.107;
   1:  PR[91,2] = PR[90,2] + 28.118;
   1:  PR[91,3] = PR[90,3] + 86.914;
   1:L PR[91] R[100]mm/sec CNT100;
   1:  PR[91,1] = PR[90,1] + 27.930;
   1:  PR[91,2] = PR[90,2] + 27.821;
   1:  PR[91,3] = PR[90,3] + 86.936;
   1:L PR[91] R[100]mm/sec CNT100;
   1:  PR[91,1] = PR[90,1] + 25.049;
   1:  PR[91,2] = PR[90,2] + 27.153;
   1:  PR[91,3] = PR[90,3] + 86.958;
   1:L PR[91] R[100]mm/sec CNT100;
   1:  PR[91,1] = PR[90,1] + 23.328;
   1:  PR[91,2] = PR[90,2] + 26.778;
   1:  PR[91,3] = PR[90,3] + 86.970;
   1:L PR[91] R[100]mm/sec CNT100;
   1:  PR[91,1] = PR[90,1] + 22.303;
   1:  PR[91,2] = PR[90,2] + 26.533;
   1:  PR[91,3] = PR[90,3] + 86.978;
   1:L PR[91] R[100]mm/sec CNT100;
   1:  PR[91,1] = PR[90,1] + 17.727;
   1:  PR[91,2] = PR[90,2] + 26.631;
   1:  PR[91,3] = PR[90,3] + 86.982;
   1:L PR[91] R[100]mm/sec CNT100;
   1:  PR[91,1] = PR[90,1] + 14.200;
   1:  PR[91,2] = PR[90,2] + 26.198;
   1:  PR[91,3] = PR[90,3] + 87.001;
   1:L PR[91] R[100]mm/sec CNT100;
   1:  PR[91,1] = PR[90,1] + 13.197;
   1:  PR[91,2] = PR[90,2] + 26.031;
   1:  PR[91,3] = PR[90,3] + 87.016;
   1:L PR[91] R[100]mm/sec CNT100;
   1:  PR[91,1] = PR[90,1] + 11.029;
   1:  PR[91,2] = PR[90,2] + 26.214;
   1:  PR[91,3] = PR[90,3] + 87.021;
   1:L PR[91] R[100]mm/sec CNT100;
   1:  PR[91,1] = PR[90,1] + 9.854;
   1:  PR[91,2] = PR[90,2] + 26.280;
   1:  PR[91,3] = PR[90,3] + 87.030;
   1:L PR[91] R[100]mm/sec CNT100;
   1:  PR[91,1] = PR[90,1] + 5.422;
   1:  PR[91,2] = PR[90,2] + 26.244;
   1:  PR[91,3] = PR[90,3] + 87.035;
   1:L PR[91] R[100]mm/sec CNT100;
   1:  PR[91,1] = PR[90,1] + 3.261;
   1:  PR[91,2] = PR[90,2] + 26.343;
   1:  PR[91,3] = PR[90,3] + 87.054;
   1:L PR[91] R[100]mm/sec CNT100;
   1:  PR[91,1] = PR[90,1] + -5.595;
   1:  PR[91,2] = PR[90,2] + 26.622;
   1:  PR[91,3] = PR[90,3] + 87.063;
   1:L PR[91] R[100]mm/sec CNT100;
   1:  PR[91,1] = PR[90,1] + -10.070;
   1:  PR[91,2] = PR[90,2] + 26.473;
   1:  PR[91,3] = PR[90,3] + 87.100;
   1:L PR[91] R[100]mm/sec CNT100;
   1:  PR[91,1] = PR[90,1] + -15.722;
   1:  PR[91,2] = PR[90,2] + 26.255;
   1:  PR[91,3] = PR[90,3] + 87.119;
   1:L PR[91] R[100]mm/sec CNT100;
   1:  PR[91,1] = PR[90,1] + -25.383;
   1:  PR[91,2] = PR[90,2] + 25.236;
   1:  PR[91,3] = PR[90,3] + 87.143;
   1:L PR[91] R[100]mm/sec CNT100;
   1:  PR[91,1] = PR[90,1] + -34.305;
   1:  PR[91,2] = PR[90,2] + 23.639;
   1:  PR[91,3] = PR[90,3] + 87.184;
   1:L PR[91] R[100]mm/sec CNT100;
   1:  PR[91,1] = PR[90,1] + -43.755;
   1:  PR[91,2] = PR[90,2] + 20.827;
   1:  PR[91,3] = PR[90,3] + 87.222;
   1:L PR[91] R[100]mm/sec CNT100;
   1:  PR[91,1] = PR[90,1] + -44.200;
   1:  PR[91,2] = PR[90,2] + 20.657;
   1:  PR[91,3] = PR[90,3] + 87.264;
   1:L PR[91] R[100]mm/sec CNT100;
   1:  PR[91,1] = PR[90,1] + -44.933;
   1:  PR[91,2] = PR[90,2] + 20.319;
   1:  PR[91,3] = PR[90,3] + 87.266;
   1:L PR[91] R[100]mm/sec CNT100;
   1:  PR[91,1] = PR[90,1] + -50.386;
   1:  PR[91,2] = PR[90,2] + 17.540;
   1:  PR[91,3] = PR[90,3] + 87.269;
   1:L PR[91] R[100]mm/sec CNT100;
   1:  PR[91] = PR[90];
   1:  PR[91,1] = PR[90,1] + -51.542;
   1:  PR[91,2] = PR[90,2] + 15.752;
   1:  PR[91,3] = PR[90,3] + 88.595;
   1:L PR[91] R[100]mm/sec CNT100;
   1:  PR[91,1] = PR[90,1] + -54.329;
   1:  PR[91,2] = PR[90,2] + 13.650;
   1:  PR[91,3] = PR[90,3] + 87.308;
   1:L PR[91] R[100]mm/sec CNT100;
   1:  PR[91,1] = PR[90,1] + -58.402;
   1:  PR[91,2] = PR[90,2] + 9.161;
   1:  PR[91,3] = PR[90,3] + 87.323;
   1:L PR[91] R[100]mm/sec CNT100;
   1:  PR[91,1] = PR[90,1] + -60.635;
   1:  PR[91,2] = PR[90,2] + 4.283;
   1:  PR[91,3] = PR[90,3] + 87.349;
   1:L PR[91] R[100]mm/sec CNT100;
   1:  PR[91,1] = PR[90,1] + -60.738;
   1:  PR[91,2] = PR[90,2] + 3.582;
   1:  PR[91,3] = PR[90,3] + 87.372;
   1:L PR[91] R[100]mm/sec CNT100;
   1:  PR[91,1] = PR[90,1] + -60.896;
   1:  PR[91,2] = PR[90,2] + 2.913;
   1:  PR[91,3] = PR[90,3] + 87.375;
   1:L PR[91] R[100]mm/sec CNT100;
   1:  PR[91,1] = PR[90,1] + -61.524;
